LIN {X 0,Y 523.99,Z 242.839,A -85,B 0,C 180,E1 -4869.261,E2 -4869.261} C_VEL
LIN {X 0,Y 523.996,Z 242.835,A -85,B 0,C 180,E1 -4871.742,E2 -4871.742} C_VEL
LIN {X 0,Y 523.98,Z 242.844,A -85,B 0,C 180,E1 -4875.051,E2 -4875.051} C_VEL
LIN {X 0,Y 523.951,Z 242.839,A -85,B 0,C 180,E1 -4877.968,E2 -4877.968} C_VEL
LIN {X 0,Y 523.96,Z 242.841,A -85,B 0,C 180,E1 -4880.409,E2 -4880.409} C_VEL
LIN {X 0,Y 523.931,Z 242.848,A -85,B 0,C 180,E1 -4882.891,E2 -4882.891} C_VEL
LIN {X 0,Y 523.97,Z 242.839,A -85,B 0,C 180,E1 -4886.019,E2 -4886.019} C_VEL
LIN {X 0,Y 523.937,Z 242.846,A -85,B 0,C 180,E1 -4888.873,E2 -4888.873} C_VEL
LIN {X 0,Y 523.909,Z 242.843,A -85,B 0,C 180,E1 -4891.543,E2 -4891.543} C_VEL
LIN {X 0,Y 523.926,Z 242.849,A -85,B 0,C 180,E1 -4894.289,E2 -4894.289} C_VEL
LIN {X 0,Y 523.896,Z 242.849,A -85,B 0,C 180,E1 -4897.131,E2 -4897.131} C_VEL
LIN {X 0,Y 523.953,Z 242.844,A -85,B 0,C 180,E1 -4900.133,E2 -4900.133} C_VEL
LIN {X 0,Y 523.911,Z 242.846,A -85,B 0,C 180,E1 -4903.166,E2 -4903.166} C_VEL
LIN {X 0,Y 523.925,Z 242.846,A -85,B 0,C 180,E1 -4905.772,E2 -4905.772} C_VEL
LIN {X 0,Y 523.906,Z 242.848,A -85,B 0,C 180,E1 -4906.926,E2 -4906.926} C_VEL
LIN {X 0,Y 523.244,Z 242.931,A -85,B 0,C 180,E1 -4907.568,E2 -4907.568} C_VEL
LIN {X 0,Y 520.414,Z 243.286,A -85,B 0,C 180,E1 -4908.61,E2 -4908.61} C_VEL
LIN {X 0,Y 518.015,Z 243.588,A -85,B 0,C 180,E1 -4909.449,E2 -4909.449} C_VEL
LIN {X 0,Y 516.976,Z 243.717,A -85,B 0,C 180,E1 -4910.097,E2 -4910.097} C_VEL
LIN {X 0,Y 516.886,Z 243.727,A -85,B 0,C 180,E1 -4910.316,E2 -4910.316} C_VEL
LIN {X 0,Y 516.95,Z 243.891,A -85,B 0,C 180,E1 -4913.2,E2 -4913.2} C_VEL
LIN {X 0,Y 518.339,Z 251.292,A -85,B 0,C 180,E1 -4914.568,E2 -4914.568} C_VEL
LIN {X 0,Y 518.054,Z 264.877,A -85,B 0,C 180,E1 -4916.905,E2 -4916.905} C_VEL
LIN {X 0,Y 517.924,Z 268.001,A -85,B 0,C 180,E1 -4917.434,E2 -4917.434} C_VEL
LIN {X 0,Y 520.396,Z 279.84,A -85,B 0,C 180,E1 -4917.697,E2 -4917.697} C_VEL
LIN {X 0,Y 519.679,Z 404.722,A -85,B 0,C 180,E1 -4919.471,E2 -4919.471} C_VEL
LIN {X 0,Y 519.41,Z 419.428,A -85,B 0,C 180,E1 -4919.847,E2 -4919.847} C_VEL
LIN {X 0,Y 519.138,Z 432.509,A -85,B 0,C 180,E1 -4920.333,E2 -4920.333} C_VEL
LIN {X 0,Y 518.762,Z 444.641,A -85,B 0,C 180,E1 -4920.921,E2 -4920.921} C_VEL
LIN {X 0,Y 518.386,Z 456.881,A -85,B 0,C 180,E1 -4921.673,E2 -4921.673} C_VEL
LIN {X 0,Y 518.005,Z 468.213,A -85,B 0,C 180,E1 -4922.53,E2 -4922.53} C_VEL
LIN {X 0,Y 517.588,Z 479.491,A -85,B 0,C 180,E1 -4923.568,E2 -4923.568} C_VEL
LIN {X 0,Y 517.236,Z 489.292,A -85,B 0,C 180,E1 -4924.659,E2 -4924.659} C_VEL
LIN {X 0,Y 516.935,Z 498.728,A -85,B 0,C 180,E1 -4925.93,E2 -4925.93} C_VEL
LIN {X 0,Y 516.671,Z 506.432,A -85,B 0,C 180,E1 -4927.191,E2 -4927.191} C_VEL
LIN {X 0,Y 516.493,Z 512.724,A -85,B 0,C 180,E1 -4928.446,E2 -4928.446} C_VEL
LIN {X 0,Y 516.401,Z 518.527,A -85,B 0,C 180,E1 -4929.889,E2 -4929.889} C_VEL
LIN {X 0,Y 516.308,Z 522.989,A -85,B 0,C 180,E1 -4931.345,E2 -4931.345} C_VEL
LIN {X 0,Y 516.228,Z 525.75,A -85,B 0,C 180,E1 -4932.572,E2 -4932.572} C_VEL
LIN {X 0,Y 516.155,Z 528.093,A -85,B 0,C 180,E1 -4934.198,E2 -4934.198} C_VEL
LIN {X 0,Y 516.233,Z 528.801,A -85,B 0,C 180,E1 -4935.141,E2 -4935.141} C_VEL
LIN {X 0,Y 516.167,Z 528.929,A -85,B 0,C 180,E1 -4936.617,E2 -4936.617} C_VEL
LIN {X 0,Y 516.222,Z 527.753,A -85,B 0,C 180,E1 -4938.217,E2 -4938.217} C_VEL
LIN {X 0,Y 516.246,Z 525.195,A -85,B 0,C 180,E1 -4939.807,E2 -4939.807} C_VEL
LIN {X 0,Y 516.343,Z 521.175,A -85,B 0,C 180,E1 -4941.389,E2 -4941.389} C_VEL
LIN {X 0,Y 516.464,Z 515.615,A -85,B 0,C 180,E1 -4942.966,E2 -4942.966} C_VEL
LIN {X 0,Y 516.564,Z 510.366,A -85,B 0,C 180,E1 -4944.144,E2 -4944.144} C_VEL
LIN {X 0,Y 516.803,Z 502.83,A -85,B 0,C 180,E1 -4945.515,E2 -4945.515} C_VEL
LIN {X 0,Y 517.05,Z 493.564,A -85,B 0,C 180,E1 -4946.883,E2 -4946.883} C_VEL
LIN {X 0,Y 517.424,Z 483.883,A -85,B 0,C 180,E1 -4948.054,E2 -4948.054} C_VEL
LIN {X 0,Y 517.772,Z 473.197,A -85,B 0,C 180,E1 -4949.125,E2 -4949.125} C_VEL
LIN {X 0,Y 518.286,Z 461.343,A -85,B 0,C 180,E1 -4950.097,E2 -4950.097} C_VEL
LIN {X 0,Y 518.658,Z 449.737,A -85,B 0,C 180,E1 -4950.874,E2 -4950.874} C_VEL
LIN {X 0,Y 519.008,Z 437.105,A -85,B 0,C 180,E1 -4951.552,E2 -4951.552} C_VEL
LIN {X 0,Y 519.332,Z 424.209,A -85,B 0,C 180,E1 -4952.084,E2 -4952.084} C_VEL
LIN {X 0,Y 519.589,Z 410.377,A -85,B 0,C 180,E1 -4952.495,E2 -4952.495} C_VEL
LIN {X 0,Y 519.741,Z 396.025,A -85,B 0,C 180,E1 -4952.761,E2 -4952.761} C_VEL
LIN {X 0,Y 520.372,Z 279.837,A -85,B 0,C 180,E1 -4954.393,E2 -4954.393} C_VEL
LIN {X 0,Y 517.927,Z 267.832,A -85,B 0,C 180,E1 -4954.67,E2 -4954.67} C_VEL
LIN {X 0,Y 518.444,Z 251.844,A -85,B 0,C 180,E1 -4957.399,E2 -4957.399} C_VEL
LIN {X 0,Y 516.951,Z 243.718,A -85,B 0,C 180,E1 -4958.896,E2 -4958.896} C_VEL
LIN {X 0,Y 516.969,Z 243.718,A -85,B 0,C 180,E1 -4961.824,E2 -4961.824} C_VEL
LIN {X 0,Y 516.93,Z 243.719,A -85,B 0,C 180,E1 -4965.147,E2 -4965.147} C_VEL
LIN {X 0,Y 516.912,Z 243.719,A -85,B 0,C 180,E1 -4968.222,E2 -4968.222} C_VEL
LIN {X 0,Y 516.899,Z 243.718,A -85,B 0,C 180,E1 -4970.702,E2 -4970.702} C_VEL
LIN {X 0,Y 516.905,Z 243.721,A -85,B 0,C 180,E1 -4974.072,E2 -4974.072} C_VEL
LIN {X 0,Y 516.917,Z 243.715,A -85,B 0,C 180,E1 -4976.658,E2 -4976.658} C_VEL
LIN {X 0,Y 516.911,Z 243.724,A -85,B 0,C 180,E1 -4979.527,E2 -4979.527} C_VEL
LIN {X 0,Y 516.887,Z 243.719,A -85,B 0,C 180,E1 -4982.545,E2 -4982.545} C_VEL
LIN {X 0,Y 516.87,Z 243.728,A -85,B 0,C 180,E1 -4985.333,E2 -4985.333} C_VEL
LIN {X 0,Y 516.868,Z 243.724,A -85,B 0,C 180,E1 -4987.944,E2 -4987.944} C_VEL
LIN {X 0,Y 516.903,Z 243.718,A -85,B 0,C 180,E1 -4990.739,E2 -4990.739} C_VEL
LIN {X 0,Y 516.869,Z 243.723,A -85,B 0,C 180,E1 -4993.903,E2 -4993.903} C_VEL
LIN {X 0,Y 516.869,Z 243.722,A -85,B 0,C 180,E1 -4996.107,E2 -4996.107} C_VEL
LIN {X 0,Y 516.894,Z 243.727,A -85,B 0,C 180,E1 -4999.261,E2 -4999.261} C_VEL
LIN {X 0,Y 516.869,Z 243.722,A -85,B 0,C 180,E1 -5002.057,E2 -5002.057} C_VEL
LIN {X 0,Y 516.884,Z 243.728,A -85,B 0,C 180,E1 -5005.177,E2 -5005.177} C_VEL
LIN {X 0,Y 516.87,Z 243.721,A -85,B 0,C 180,E1 -5007.977,E2 -5007.977} C_VEL
LIN {X 0,Y 516.923,Z 243.719,A -85,B 0,C 180,E1 -5010.697,E2 -5010.697} C_VEL
LIN {X 0,Y 516.932,Z 243.714,A -85,B 0,C 180,E1 -5013.804,E2 -5013.804} C_VEL
LIN {X 0,Y 516.86,Z 243.73,A -85,B 0,C 180,E1 -5016.777,E2 -5016.777} C_VEL
LIN {X 0,Y 516.928,Z 243.714,A -85,B 0,C 180,E1 -5019.732,E2 -5019.732} C_VEL
LIN {X 0,Y 516.92,Z 243.721,A -85,B 0,C 180,E1 -5022.597,E2 -5022.597} C_VEL
LIN {X 0,Y 516.931,Z 243.719,A -85,B 0,C 180,E1 -5025.031,E2 -5025.031} C_VEL
LIN {X 0,Y 516.955,Z 243.713,A -85,B 0,C 180,E1 -5028.235,E2 -5028.235} C_VEL
LIN {X 0,Y 516.961,Z 243.711,A -85,B 0,C 180,E1 -5031.401,E2 -5031.401} C_VEL
LIN {X 0,Y 517.001,Z 243.705,A -85,B 0,C 180,E1 -5033.758,E2 -5033.758} C_VEL
LIN {X 0,Y 517.008,Z 243.708,A -85,B 0,C 180,E1 -5036.884,E2 -5036.884} C_VEL
LIN {X 0,Y 517.076,Z 243.698,A -85,B 0,C 180,E1 -5040.001,E2 -5040.001} C_VEL
LIN {X 0,Y 517.008,Z 243.705,A -85,B 0,C 180,E1 -5043.118,E2 -5043.118} C_VEL
LIN {X 0,Y 517.003,Z 243.712,A -85,B 0,C 180,E1 -5046.244,E2 -5046.244} C_VEL
LIN {X 0,Y 516.948,Z 243.712,A -85,B 0,C 180,E1 -5049.39,E2 -5049.39} C_VEL
LIN {X 0,Y 516.945,Z 243.715,A -85,B 0,C 180,E1 -5051.808,E2 -5051.808} C_VEL
LIN {X 0,Y 516.938,Z 243.713,A -85,B 0,C 180,E1 -5055.147,E2 -5055.147} C_VEL
LIN {X 0,Y 516.92,Z 243.723,A -85,B 0,C 180,E1 -5058.223,E2 -5058.223} C_VEL
LIN {X 0,Y 516.907,Z 243.718,A -85,B 0,C 180,E1 -5060.703,E2 -5060.703} C_VEL
LIN {X 0,Y 516.906,Z 243.726,A -85,B 0,C 180,E1 -5064.073,E2 -5064.073} C_VEL
LIN {X 0,Y 516.922,Z 243.716,A -85,B 0,C 180,E1 -5066.659,E2 -5066.659} C_VEL
LIN {X 0,Y 516.916,Z 243.719,A -85,B 0,C 180,E1 -5069.527,E2 -5069.527} C_VEL
LIN {X 0,Y 516.897,Z 243.719,A -85,B 0,C 180,E1 -5072.545,E2 -5072.545} C_VEL
LIN {X 0,Y 516.88,Z 243.722,A -85,B 0,C 180,E1 -5075.333,E2 -5075.333} C_VEL
LIN {X 0,Y 516.879,Z 243.727,A -85,B 0,C 180,E1 -5077.944,E2 -5077.944} C_VEL
LIN {X 0,Y 516.882,Z 243.72,A -85,B 0,C 180,E1 -5080.743,E2 -5080.743} C_VEL
LIN {X 0,Y 516.881,Z 243.72,A -85,B 0,C 180,E1 -5082.832,E2 -5082.832} C_VEL
LIN {X 0,Y 516.922,Z 243.716,A -85,B 0,C 180,E1 -5085.011,E2 -5085.011} C_VEL
LIN {X 0,Y 516.914,Z 243.716,A -85,B 0,C 180,E1 -5088.399,E2 -5088.399} C_VEL
LIN {X 0,Y 516.879,Z 243.725,A -85,B 0,C 180,E1 -5091.285,E2 -5091.285} C_VEL
LIN {X 0,Y 516.871,Z 243.722,A -85,B 0,C 180,E1 -5094.22,E2 -5094.22} C_VEL
LIN {X 0,Y 516.896,Z 243.721,A -85,B 0,C 180,E1 -5097.054,E2 -5097.054} C_VEL
LIN {X 0,Y 516.893,Z 243.726,A -85,B 0,C 180,E1 -5099.797,E2 -5099.797} C_VEL
LIN {X 0,Y 516.927,Z 243.719,A -85,B 0,C 180,E1 -5102.468,E2 -5102.468} C_VEL
LIN {X 0,Y 516.964,Z 243.89,A -85,B 0,C 180,E1 -5103.85,E2 -5103.85} C_VEL
LIN {X 0,Y 519.153,Z 254.919,A -85,B 0,C 180,E1 -5105.614,E2 -5105.614} C_VEL
LIN {X 0,Y 518.575,Z 273.415,A -85,B 0,C 180,E1 -5108.328,E2 -5108.328} C_VEL
LIN {X 0,Y 517.999,Z 294.61,A -85,B 0,C 180,E1 -5111.378,E2 -5111.378} C_VEL
LIN {X 0,Y 520.416,Z 308.774,A -85,B 0,C 180,E1 -5111.669,E2 -5111.669} C_VEL
LIN {X 0,Y 519.645,Z 432.714,A -85,B 0,C 180,E1 -5113.424,E2 -5113.424} C_VEL
LIN {X 0,Y 519.343,Z 447.15,A -85,B 0,C 180,E1 -5113.788,E2 -5113.788} C_VEL
LIN {X 0,Y 519.065,Z 460.688,A -85,B 0,C 180,E1 -5114.289,E2 -5114.289} C_VEL
LIN {X 0,Y 518.676,Z 472.91,A -85,B 0,C 180,E1 -5114.881,E2 -5114.881} C_VEL
LIN {X 0,Y 518.248,Z 485.767,A -85,B 0,C 180,E1 -5115.671,E2 -5115.671} C_VEL
LIN {X 0,Y 517.847,Z 497.459,A -85,B 0,C 180,E1 -5116.561,E2 -5116.561} C_VEL
LIN {X 0,Y 517.494,Z 507.19,A -85,B 0,C 180,E1 -5117.45,E2 -5117.45} C_VEL
LIN {X 0,Y 517.141,Z 517.972,A -85,B 0,C 180,E1 -5118.635,E2 -5118.635} C_VEL
LIN {X 0,Y 516.832,Z 526.875,A -85,B 0,C 180,E1 -5119.818,E2 -5119.818} C_VEL
LIN {X 0,Y 516.615,Z 535.409,A -85,B 0,C 180,E1 -5121.197,E2 -5121.197} C_VEL
LIN {X 0,Y 516.447,Z 542.287,A -85,B 0,C 180,E1 -5122.572,E2 -5122.572} C_VEL
LIN {X 0,Y 516.372,Z 547.028,A -85,B 0,C 180,E1 -5123.749,E2 -5123.749} C_VEL
LIN {X 0,Y 516.306,Z 550.868,A -85,B 0,C 180,E1 -5124.924,E2 -5124.924} C_VEL
LIN {X 0,Y 516.325,Z 553.828,A -85,B 0,C 180,E1 -5126.098,E2 -5126.098} C_VEL
LIN {X 0,Y 516.26,Z 556.535,A -85,B 0,C 180,E1 -5127.659,E2 -5127.659} C_VEL
LIN {X 0,Y 516.158,Z 557.874,A -85,B 0,C 180,E1 -5129.22,E2 -5129.22} C_VEL
LIN {X 0,Y 516.158,Z 557.873,A -85,B 0,C 180,E1 -5130.78,E2 -5130.78} C_VEL
LIN {X 0,Y 516.26,Z 556.534,A -85,B 0,C 180,E1 -5132.34,E2 -5132.34} C_VEL
LIN {X 0,Y 516.325,Z 553.826,A -85,B 0,C 180,E1 -5133.902,E2 -5133.902} C_VEL
LIN {X 0,Y 516.361,Z 549.672,A -85,B 0,C 180,E1 -5135.467,E2 -5135.467} C_VEL
LIN {X 0,Y 516.403,Z 543.949,A -85,B 0,C 180,E1 -5137.035,E2 -5137.035} C_VEL
LIN {X 0,Y 516.578,Z 537.501,A -85,B 0,C 180,E1 -5138.41,E2 -5138.41} C_VEL
LIN {X 0,Y 516.765,Z 529.489,A -85,B 0,C 180,E1 -5139.788,E2 -5139.788} C_VEL
LIN {X 0,Y 517.067,Z 521.112,A -85,B 0,C 180,E1 -5140.969,E2 -5140.969} C_VEL
LIN {X 0,Y 517.378,Z 510.785,A -85,B 0,C 180,E1 -5142.181,E2 -5142.181} C_VEL
LIN {X 0,Y 517.749,Z 499.776,A -85,B 0,C 180,E1 -5143.242,E2 -5143.242} C_VEL
LIN {X 0,Y 518.138,Z 488.589,A -85,B 0,C 180,E1 -5144.131,E2 -5144.131} C_VEL
LIN {X 0,Y 518.532,Z 476.405,A -85,B 0,C 180,E1 -5144.922,E2 -5144.922} C_VEL
LIN {X 0,Y 518.986,Z 462.889,A -85,B 0,C 180,E1 -5145.613,E2 -5145.613} C_VEL
LIN {X 0,Y 519.284,Z 448.75,A -85,B 0,C 180,E1 -5146.158,E2 -5146.158} C_VEL
LIN {X 0,Y 519.589,Z 434.929,A -85,B 0,C 180,E1 -5146.527,E2 -5146.527} C_VEL
LIN {X 0,Y 519.753,Z 412.74,A -85,B 0,C 180,E1 -5146.875,E2 -5146.875} C_VEL
LIN {X 0,Y 520.29,Z 307.794,A -85,B 0,C 180,E1 -5148.349,E2 -5148.349} C_VEL
LIN {X 0,Y 518.005,Z 294.369,A -85,B 0,C 180,E1 -5148.633,E2 -5148.633} C_VEL
LIN {X 0,Y 518.604,Z 271.897,A -85,B 0,C 180,E1 -5151.88,E2 -5151.88} C_VEL
LIN {X 0,Y 519.14,Z 254.866,A -85,B 0,C 180,E1 -5154.387,E2 -5154.387} C_VEL
LIN {X 0,Y 516.931,Z 243.722,A -85,B 0,C 180,E1 -5156.192,E2 -5156.192} C_VEL
LIN {X 0,Y 516.922,Z 243.719,A -85,B 0,C 180,E1 -5159.304,E2 -5159.304} C_VEL
LIN {X 0,Y 516.897,Z 243.726,A -85,B 0,C 180,E1 -5162.543,E2 -5162.543} C_VEL
LIN {X 0,Y 516.865,Z 243.726,A -85,B 0,C 180,E1 -5165.329,E2 -5165.329} C_VEL
LIN {X 0,Y 516.879,Z 243.724,A -85,B 0,C 180,E1 -5167.942,E2 -5167.942} C_VEL
LIN {X 0,Y 516.882,Z 243.723,A -85,B 0,C 180,E1 -5170.741,E2 -5170.741} C_VEL
LIN {X 0,Y 516.902,Z 243.721,A -85,B 0,C 180,E1 -5172.828,E2 -5172.828} C_VEL
LIN {X 0,Y 516.92,Z 243.716,A -85,B 0,C 180,E1 -5175.009,E2 -5175.009} C_VEL
LIN {X 0,Y 516.914,Z 243.723,A -85,B 0,C 180,E1 -5178.397,E2 -5178.397} C_VEL
LIN {X 0,Y 516.879,Z 243.721,A -85,B 0,C 180,E1 -5181.283,E2 -5181.283} C_VEL
LIN {X 0,Y 516.887,Z 243.718,A -85,B 0,C 180,E1 -5184.22,E2 -5184.22} C_VEL
LIN {X 0,Y 516.893,Z 243.719,A -85,B 0,C 180,E1 -5187.052,E2 -5187.052} C_VEL
LIN {X 0,Y 516.896,Z 243.723,A -85,B 0,C 180,E1 -5189.796,E2 -5189.796} C_VEL
LIN {X 0,Y 516.923,Z 243.716,A -85,B 0,C 180,E1 -5192.466,E2 -5192.466} C_VEL
LIN {X 0,Y 516.904,Z 243.718,A -85,B 0,C 180,E1 -5195.071,E2 -5195.071} C_VEL
LIN {X 0,Y 516.863,Z 243.729,A -85,B 0,C 180,E1 -5197.62,E2 -5197.62} C_VEL
LIN {X 0,Y 516.925,Z 243.717,A -85,B 0,C 180,E1 -5200.129,E2 -5200.129} C_VEL
LIN {X 0,Y 516.924,Z 243.715,A -85,B 0,C 180,E1 -5202.595,E2 -5202.595} C_VEL
LIN {X 0,Y 516.934,Z 243.714,A -85,B 0,C 180,E1 -5205.029,E2 -5205.029} C_VEL
LIN {X 0,Y 516.957,Z 243.709,A -85,B 0,C 180,E1 -5208.233,E2 -5208.233} C_VEL
LIN {X 0,Y 516.964,Z 243.718,A -85,B 0,C 180,E1 -5211.399,E2 -5211.399} C_VEL
LIN {X 0,Y 517.001,Z 243.71,A -85,B 0,C 180,E1 -5213.756,E2 -5213.756} C_VEL
LIN {X 0,Y 517.007,Z 243.706,A -85,B 0,C 180,E1 -5216.882,E2 -5216.882} C_VEL
LIN {X 0,Y 517.072,Z 243.697,A -85,B 0,C 180,E1 -5219.999,E2 -5219.999} C_VEL
LIN {X 0,Y 517.007,Z 243.711,A -85,B 0,C 180,E1 -5223.116,E2 -5223.116} C_VEL
LIN {X 0,Y 516.999,Z 243.704,A -85,B 0,C 180,E1 -5226.242,E2 -5226.242} C_VEL
LIN {X 0,Y 516.945,Z 243.715,A -85,B 0,C 180,E1 -5229.388,E2 -5229.388} C_VEL
LIN {X 0,Y 516.945,Z 243.713,A -85,B 0,C 180,E1 -5231.809,E2 -5231.809} C_VEL
LIN {X 0,Y 516.931,Z 243.721,A -85,B 0,C 180,E1 -5235.145,E2 -5235.145} C_VEL
LIN {X 0,Y 516.912,Z 243.717,A -85,B 0,C 180,E1 -5238.221,E2 -5238.221} C_VEL
LIN {X 0,Y 516.902,Z 243.724,A -85,B 0,C 180,E1 -5240.7,E2 -5240.7} C_VEL
LIN {X 0,Y 516.878,Z 243.722,A -85,B 0,C 180,E1 -5243.222,E2 -5243.222} C_VEL
LIN {X 0,Y 516.928,Z 243.717,A -85,B 0,C 180,E1 -5246.195,E2 -5246.195} C_VEL
LIN {X 0,Y 516.922,Z 243.715,A -85,B 0,C 180,E1 -5249.303,E2 -5249.303} C_VEL
LIN {X 0,Y 516.882,Z 243.727,A -85,B 0,C 180,E1 -5252.543,E2 -5252.543} C_VEL
LIN {X 0,Y 516.865,Z 243.72,A -85,B 0,C 180,E1 -5255.331,E2 -5255.331} C_VEL
LIN {X 0,Y 516.867,Z 243.726,A -85,B 0,C 180,E1 -5257.943,E2 -5257.943} C_VEL
LIN {X 0,Y 516.889,Z 243.724,A -85,B 0,C 180,E1 -5260.739,E2 -5260.739} C_VEL
LIN {X 0,Y 516.867,Z 243.727,A -85,B 0,C 180,E1 -5263.903,E2 -5263.903} C_VEL
LIN {X 0,Y 516.867,Z 243.73,A -85,B 0,C 180,E1 -5266.106,E2 -5266.106} C_VEL
LIN {X 0,Y 516.889,Z 243.722,A -85,B 0,C 180,E1 -5269.26,E2 -5269.26} C_VEL
LIN {X 0,Y 516.886,Z 243.727,A -85,B 0,C 180,E1 -5270.316,E2 -5270.316} C_VEL
LIN {X 0,Y 516.194,Z 243.813,A -85,B 0,C 180,E1 -5270.75,E2 -5270.75} C_VEL
LIN {X 0,Y 513.334,Z 244.168,A -85,B 0,C 180,E1 -5271.428,E2 -5271.428} C_VEL
LIN {X 0,Y 510.486,Z 244.526,A -85,B 0,C 180,E1 -5272.113,E2 -5272.113} C_VEL
LIN {X 0,Y 509.827,Z 244.607,A -85,B 0,C 180,E1 -5272.555,E2 -5272.555} C_VEL
LIN {X 0,Y 509.854,Z 244.69,A -85,B 0,C 180,E1 -5272.965,E2 -5272.965} C_VEL
LIN {X 0,Y 511.436,Z 252.766,A -85,B 0,C 180,E1 -5274.488,E2 -5274.488} C_VEL
LIN {X 0,Y 511.043,Z 267.316,A -85,B 0,C 180,E1 -5277.02,E2 -5277.02} C_VEL
LIN {X 0,Y 511.057,Z 268.302,A -85,B 0,C 180,E1 -5277.175,E2 -5277.175} C_VEL
LIN {X 0,Y 513.655,Z 280.569,A -85,B 0,C 180,E1 -5277.455,E2 -5277.455} C_VEL
LIN {X 0,Y 512.898,Z 405.162,A -85,B 0,C 180,E1 -5279.252,E2 -5279.252} C_VEL
LIN {X 0,Y 512.592,Z 419.721,A -85,B 0,C 180,E1 -5279.629,E2 -5279.629} C_VEL
LIN {X 0,Y 512.304,Z 432.99,A -85,B 0,C 180,E1 -5280.131,E2 -5280.131} C_VEL
LIN {X 0,Y 511.912,Z 444.924,A -85,B 0,C 180,E1 -5280.72,E2 -5280.72} C_VEL
LIN {X 0,Y 511.509,Z 456.973,A -85,B 0,C 180,E1 -5281.469,E2 -5281.469} C_VEL
LIN {X 0,Y 511.073,Z 468.458,A -85,B 0,C 180,E1 -5282.348,E2 -5282.348} C_VEL
LIN {X 0,Y 510.603,Z 480.329,A -85,B 0,C 180,E1 -5283.462,E2 -5283.462} C_VEL
LIN {X 0,Y 510.182,Z 491.265,A -85,B 0,C 180,E1 -5284.721,E2 -5284.721} C_VEL
LIN {X 0,Y 509.866,Z 500.381,A -85,B 0,C 180,E1 -5286.007,E2 -5286.007} C_VEL
LIN {X 0,Y 509.612,Z 507.829,A -85,B 0,C 180,E1 -5287.286,E2 -5287.286} C_VEL
LIN {X 0,Y 509.413,Z 513.899,A -85,B 0,C 180,E1 -5288.556,E2 -5288.556} C_VEL
LIN {X 0,Y 509.328,Z 518.789,A -85,B 0,C 180,E1 -5289.821,E2 -5289.821} C_VEL
LIN {X 0,Y 509.242,Z 522.647,A -85,B 0,C 180,E1 -5291.076,E2 -5291.076} C_VEL
LIN {X 0,Y 509.15,Z 525.583,A -85,B 0,C 180,E1 -5292.322,E2 -5292.322} C_VEL
LIN {X 0,Y 509.058,Z 528.092,A -85,B 0,C 180,E1 -5293.972,E2 -5293.972} C_VEL
LIN {X 0,Y 509.113,Z 529.158,A -85,B 0,C 180,E1 -5295.613,E2 -5295.613} C_VEL
LIN {X 0,Y 509.089,Z 528.831,A -85,B 0,C 180,E1 -5297.24,E2 -5297.24} C_VEL
LIN {X 0,Y 509.175,Z 527.124,A -85,B 0,C 180,E1 -5298.859,E2 -5298.859} C_VEL
LIN {X 0,Y 509.144,Z 524.041,A -85,B 0,C 180,E1 -5300.466,E2 -5300.466} C_VEL
LIN {X 0,Y 509.31,Z 519.482,A -85,B 0,C 180,E1 -5302.069,E2 -5302.069} C_VEL
LIN {X 0,Y 509.461,Z 513.286,A -85,B 0,C 180,E1 -5303.664,E2 -5303.664} C_VEL
LIN {X 0,Y 509.618,Z 506.418,A -85,B 0,C 180,E1 -5305.056,E2 -5305.056} C_VEL
LIN {X 0,Y 509.871,Z 497.941,A -85,B 0,C 180,E1 -5306.444,E2 -5306.444} C_VEL
LIN {X 0,Y 510.257,Z 489.099,A -85,B 0,C 180,E1 -5307.632,E2 -5307.632} C_VEL
LIN {X 0,Y 510.66,Z 478.455,A -85,B 0,C 180,E1 -5308.817,E2 -5308.817} C_VEL
LIN {X 0,Y 511.131,Z 467.685,A -85,B 0,C 180,E1 -5309.803,E2 -5309.803} C_VEL
LIN {X 0,Y 511.564,Z 455.947,A -85,B 0,C 180,E1 -5310.689,E2 -5310.689} C_VEL
LIN {X 0,Y 512.024,Z 442.98,A -85,B 0,C 180,E1 -5311.475,E2 -5311.475} C_VEL
LIN {X 0,Y 512.39,Z 429.328,A -85,B 0,C 180,E1 -5312.113,E2 -5312.113} C_VEL
LIN {X 0,Y 512.707,Z 414.894,A -85,B 0,C 180,E1 -5312.603,E2 -5312.603} C_VEL
LIN {X 0,Y 512.913,Z 400.49,A -85,B 0,C 180,E1 -5312.921,E2 -5312.921} C_VEL
LIN {X 0,Y 513.709,Z 281.236,A -85,B 0,C 180,E1 -5314.622,E2 -5314.622} C_VEL
LIN {X 0,Y 510.972,Z 268.014,A -85,B 0,C 180,E1 -5314.931,E2 -5314.931} C_VEL
LIN {X 0,Y 511.507,Z 253.142,A -85,B 0,C 180,E1 -5317.5,E2 -5317.5} C_VEL
LIN {X 0,Y 509.938,Z 244.592,A -85,B 0,C 180,E1 -5319.119,E2 -5319.119} C_VEL
LIN {X 0,Y 509.937,Z 244.595,A -85,B 0,C 180,E1 -5321.931,E2 -5321.931} C_VEL
LIN {X 0,Y 509.879,Z 244.598,A -85,B 0,C 180,E1 -5325.242,E2 -5325.242} C_VEL
LIN {X 0,Y 509.874,Z 244.599,A -85,B 0,C 180,E1 -5328.001,E2 -5328.001} C_VEL
LIN {X 0,Y 509.837,Z 244.598,A -85,B 0,C 180,E1 -5331.002,E2 -5331.002} C_VEL
LIN {X 0,Y 509.828,Z 244.605,A -85,B 0,C 180,E1 -5333.563,E2 -5333.563} C_VEL
LIN {X 0,Y 509.902,Z 244.59,A -85,B 0,C 180,E1 -5336.38,E2 -5336.38} C_VEL
LIN {X 0,Y 509.872,Z 244.594,A -85,B 0,C 180,E1 -5338.844,E2 -5338.844} C_VEL
LIN {X 0,Y 509.813,Z 244.609,A -85,B 0,C 180,E1 -5341.59,E2 -5341.59} C_VEL
LIN {X 0,Y 509.841,Z 244.597,A -85,B 0,C 180,E1 -5344.414,E2 -5344.414} C_VEL
LIN {X 0,Y 509.805,Z 244.609,A -85,B 0,C 180,E1 -5347.341,E2 -5347.341} C_VEL
LIN {X 0,Y 509.865,Z 244.594,A -85,B 0,C 180,E1 -5350.379,E2 -5350.379} C_VEL
LIN {X 0,Y 509.827,Z 244.603,A -85,B 0,C 180,E1 -5353.065,E2 -5353.065} C_VEL
LIN {X 0,Y 509.817,Z 244.602,A -85,B 0,C 180,E1 -5355.793,E2 -5355.793} C_VEL
LIN {X 0,Y 509.857,Z 244.596,A -85,B 0,C 180,E1 -5358.577,E2 -5358.577} C_VEL
LIN {X 0,Y 509.843,Z 244.598,A -85,B 0,C 180,E1 -5361.786,E2 -5361.786} C_VEL
LIN {X 0,Y 509.834,Z 244.6,A -85,B 0,C 180,E1 -5364.624,E2 -5364.624} C_VEL
LIN {X 0,Y 509.853,Z 244.599,A -85,B 0,C 180,E1 -5367.482,E2 -5367.482} C_VEL
LIN {X 0,Y 509.869,Z 244.594,A -85,B 0,C 180,E1 -5370.27,E2 -5370.27} C_VEL
LIN {X 0,Y 509.876,Z 244.601,A -85,B 0,C 180,E1 -5372.945,E2 -5372.945} C_VEL
LIN {X 0,Y 509.858,Z 244.596,A -85,B 0,C 180,E1 -5375.575,E2 -5375.575} C_VEL
LIN {X 0,Y 509.811,Z 244.601,A -85,B 0,C 180,E1 -5378.15,E2 -5378.15} C_VEL
LIN {X 0,Y 509.854,Z 244.602,A -85,B 0,C 180,E1 -5380.683,E2 -5380.683} C_VEL
LIN {X 0,Y 509.876,Z 244.596,A -85,B 0,C 180,E1 -5383.176,E2 -5383.176} C_VEL
LIN {X 0,Y 509.854,Z 244.595,A -85,B 0,C 180,E1 -5385.635,E2 -5385.635} C_VEL
LIN {X 0,Y 509.891,Z 244.592,A -85,B 0,C 180,E1 -5388.124,E2 -5388.124} C_VEL
LIN {X 0,Y 509.907,Z 244.59,A -85,B 0,C 180,E1 -5391.281,E2 -5391.281} C_VEL
LIN {X 0,Y 509.969,Z 244.581,A -85,B 0,C 180,E1 -5393.671,E2 -5393.671} C_VEL
LIN {X 0,Y 510.047,Z 244.571,A -85,B 0,C 180,E1 -5397.632,E2 -5397.632} C_VEL
LIN {X 0,Y 510.057,Z 244.574,A -85,B 0,C 180,E1 -5400.791,E2 -5400.791} C_VEL
LIN {X 0,Y 509.95,Z 244.584,A -85,B 0,C 180,E1 -5403.161,E2 -5403.161} C_VEL
LIN {X 0,Y 509.971,Z 244.589,A -85,B 0,C 180,E1 -5406.331,E2 -5406.331} C_VEL
LIN {X 0,Y 509.909,Z 244.592,A -85,B 0,C 180,E1 -5408.721,E2 -5408.721} C_VEL
LIN {X 0,Y 509.897,Z 244.594,A -85,B 0,C 180,E1 -5411.933,E2 -5411.933} C_VEL
LIN {X 0,Y 509.887,Z 244.591,A -85,B 0,C 180,E1 -5415.243,E2 -5415.243} C_VEL
LIN {X 0,Y 509.883,Z 244.598,A -85,B 0,C 180,E1 -5418.002,E2 -5418.002} C_VEL
LIN {X 0,Y 509.845,Z 244.597,A -85,B 0,C 180,E1 -5421.003,E2 -5421.003} C_VEL
LIN {X 0,Y 509.865,Z 244.597,A -85,B 0,C 180,E1 -5424.427,E2 -5424.427} C_VEL
LIN {X 0,Y 509.881,Z 244.592,A -85,B 0,C 180,E1 -5427.057,E2 -5427.057} C_VEL
LIN {X 0,Y 509.877,Z 244.598,A -85,B 0,C 180,E1 -5429.751,E2 -5429.751} C_VEL
LIN {X 0,Y 509.873,Z 244.593,A -85,B 0,C 180,E1 -5432.776,E2 -5432.776} C_VEL
LIN {X 0,Y 509.839,Z 244.602,A -85,B 0,C 180,E1 -5435.582,E2 -5435.582} C_VEL
LIN {X 0,Y 509.848,Z 244.598,A -85,B 0,C 180,E1 -5438.339,E2 -5438.339} C_VEL
LIN {X 0,Y 509.854,Z 244.6,A -85,B 0,C 180,E1 -5441.426,E2 -5441.426} C_VEL
LIN {X 0,Y 509.855,Z 244.595,A -85,B 0,C 180,E1 -5444.669,E2 -5444.669} C_VEL
LIN {X 0,Y 509.856,Z 244.597,A -85,B 0,C 180,E1 -5448.104,E2 -5448.104} C_VEL
LIN {X 0,Y 509.845,Z 244.596,A -85,B 0,C 180,E1 -5450.648,E2 -5450.648} C_VEL
LIN {X 0,Y 509.824,Z 244.606,A -85,B 0,C 180,E1 -5453.648,E2 -5453.648} C_VEL
LIN {X 0,Y 509.86,Z 244.595,A -85,B 0,C 180,E1 -5456.54,E2 -5456.54} C_VEL
LIN {X 0,Y 509.846,Z 244.606,A -85,B 0,C 180,E1 -5459.335,E2 -5459.335} C_VEL
LIN {X 0,Y 509.893,Z 244.596,A -85,B 0,C 180,E1 -5462.055,E2 -5462.055} C_VEL
LIN {X 0,Y 509.913,Z 244.693,A -85,B 0,C 180,E1 -5463.622,E2 -5463.622} C_VEL
LIN {X 0,Y 512.268,Z 256.398,A -85,B 0,C 180,E1 -5465.521,E2 -5465.521} C_VEL
LIN {X 0,Y 511.568,Z 276.065,A -85,B 0,C 180,E1 -5468.439,E2 -5468.439} C_VEL
LIN {X 0,Y 511.047,Z 294.357,A -85,B 0,C 180,E1 -5471.114,E2 -5471.114} C_VEL
LIN {X 0,Y 513.681,Z 309.516,A -85,B 0,C 180,E1 -5471.433,E2 -5471.433} C_VEL
LIN {X 0,Y 512.849,Z 432.47,A -85,B 0,C 180,E1 -5473.198,E2 -5473.198} C_VEL
LIN {X 0,Y 512.534,Z 446.636,A -85,B 0,C 180,E1 -5473.557,E2 -5473.557} C_VEL
LIN {X 0,Y 512.224,Z 460.467,A -85,B 0,C 180,E1 -5474.073,E2 -5474.073} C_VEL
LIN {X 0,Y 511.735,Z 474.464,A -85,B 0,C 180,E1 -5474.773,E2 -5474.773} C_VEL
LIN {X 0,Y 511.28,Z 486.985,A -85,B 0,C 180,E1 -5475.573,E2 -5475.573} C_VEL
LIN {X 0,Y 510.85,Z 498.427,A -85,B 0,C 180,E1 -5476.475,E2 -5476.475} C_VEL
LIN {X 0,Y 510.441,Z 509.138,A -85,B 0,C 180,E1 -5477.496,E2 -5477.496} C_VEL
LIN {X 0,Y 510.103,Z 519.403,A -85,B 0,C 180,E1 -5478.678,E2 -5478.678} C_VEL
LIN {X 0,Y 509.741,Z 528.033,A -85,B 0,C 180,E1 -5479.876,E2 -5479.876} C_VEL
LIN {X 0,Y 509.528,Z 536.301,A -85,B 0,C 180,E1 -5481.273,E2 -5481.273} C_VEL
LIN {X 0,Y 509.37,Z 542.085,A -85,B 0,C 180,E1 -5482.468,E2 -5482.468} C_VEL
LIN {X 0,Y 509.289,Z 546.828,A -85,B 0,C 180,E1 -5483.662,E2 -5483.662} C_VEL
LIN {X 0,Y 509.235,Z 550.669,A -85,B 0,C 180,E1 -5484.853,E2 -5484.853} C_VEL
LIN {X 0,Y 509.218,Z 553.628,A -85,B 0,C 180,E1 -5486.043,E2 -5486.043} C_VEL
LIN {X 0,Y 509.189,Z 556.336,A -85,B 0,C 180,E1 -5487.627,E2 -5487.627} C_VEL
LIN {X 0,Y 509.071,Z 557.675,A -85,B 0,C 180,E1 -5489.209,E2 -5489.209} C_VEL
LIN {X 0,Y 509.071,Z 557.673,A -85,B 0,C 180,E1 -5490.791,E2 -5490.791} C_VEL
LIN {X 0,Y 509.189,Z 556.334,A -85,B 0,C 180,E1 -5492.373,E2 -5492.373} C_VEL
LIN {X 0,Y 509.217,Z 553.623,A -85,B 0,C 180,E1 -5493.957,E2 -5493.957} C_VEL
LIN {X 0,Y 509.277,Z 549.468,A -85,B 0,C 180,E1 -5495.543,E2 -5495.543} C_VEL
LIN {X 0,Y 509.328,Z 543.743,A -85,B 0,C 180,E1 -5497.134,E2 -5497.134} C_VEL
LIN {X 0,Y 509.499,Z 537.292,A -85,B 0,C 180,E1 -5498.527,E2 -5498.527} C_VEL
LIN {X 0,Y 509.719,Z 529.278,A -85,B 0,C 180,E1 -5499.924,E2 -5499.924} C_VEL
LIN {X 0,Y 510.036,Z 520.899,A -85,B 0,C 180,E1 -5501.122,E2 -5501.122} C_VEL
LIN {X 0,Y 510.398,Z 510.169,A -85,B 0,C 180,E1 -5502.394,E2 -5502.394} C_VEL
LIN {X 0,Y 510.779,Z 499.556,A -85,B 0,C 180,E1 -5503.426,E2 -5503.426} C_VEL
LIN {X 0,Y 511.225,Z 488.366,A -85,B 0,C 180,E1 -5504.326,E2 -5504.326} C_VEL
LIN {X 0,Y 511.633,Z 476.176,A -85,B 0,C 180,E1 -5505.128,E2 -5505.128} C_VEL
LIN {X 0,Y 512.147,Z 462.655,A -85,B 0,C 180,E1 -5505.827,E2 -5505.827} C_VEL
LIN {X 0,Y 512.473,Z 448.51,A -85,B 0,C 180,E1 -5506.379,E2 -5506.379} C_VEL
LIN {X 0,Y 512.791,Z 434.669,A -85,B 0,C 180,E1 -5506.752,E2 -5506.752} C_VEL
LIN {X 0,Y 512.955,Z 412.454,A -85,B 0,C 180,E1 -5507.106,E2 -5507.106} C_VEL
LIN {X 0,Y 513.621,Z 309.15,A -85,B 0,C 180,E1 -5508.573,E2 -5508.573} C_VEL
LIN {X 0,Y 511.038,Z 294.168,A -85,B 0,C 180,E1 -5508.897,E2 -5508.897} C_VEL
LIN {X 0,Y 511.687,Z 273.161,A -85,B 0,C 180,E1 -5511.979,E2 -5511.979} C_VEL
LIN {X 0,Y 512.262,Z 256.444,A -85,B 0,C 180,E1 -5514.479,E2 -5514.479} C_VEL
LIN {X 0,Y 510.248,Z 246.262,A -85,B 0,C 180,E1 -5516.151,E2 -5516.151} C_VEL
LIN {X 0,Y 509.886,Z 244.598,A -85,B 0,C 180,E1 -5516.435,E2 -5516.435} C_VEL
LIN {X 0,Y 509.877,Z 244.599,A -85,B 0,C 180,E1 -5518.843,E2 -5518.843} C_VEL
LIN {X 0,Y 509.821,Z 244.604,A -85,B 0,C 180,E1 -5521.589,E2 -5521.589} C_VEL
LIN {X 0,Y 509.847,Z 244.605,A -85,B 0,C 180,E1 -5524.413,E2 -5524.413} C_VEL
LIN {X 0,Y 509.815,Z 244.602,A -85,B 0,C 180,E1 -5527.34,E2 -5527.34} C_VEL
LIN {X 0,Y 509.836,Z 244.603,A -85,B 0,C 180,E1 -5530.381,E2 -5530.381} C_VEL
LIN {X 0,Y 509.837,Z 244.599,A -85,B 0,C 180,E1 -5533.063,E2 -5533.063} C_VEL
LIN {X 0,Y 509.828,Z 244.602,A -85,B 0,C 180,E1 -5535.791,E2 -5535.791} C_VEL
LIN {X 0,Y 509.855,Z 244.6,A -85,B 0,C 180,E1 -5538.574,E2 -5538.574} C_VEL
LIN {X 0,Y 509.848,Z 244.601,A -85,B 0,C 180,E1 -5541.785,E2 -5541.785} C_VEL
LIN {X 0,Y 509.842,Z 244.593,A -85,B 0,C 180,E1 -5544.622,E2 -5544.622} C_VEL
LIN {X 0,Y 509.861,Z 244.597,A -85,B 0,C 180,E1 -5547.48,E2 -5547.48} C_VEL
LIN {X 0,Y 509.876,Z 244.597,A -85,B 0,C 180,E1 -5550.268,E2 -5550.268} C_VEL
LIN {X 0,Y 509.88,Z 244.591,A -85,B 0,C 180,E1 -5552.943,E2 -5552.943} C_VEL
LIN {X 0,Y 509.863,Z 244.6,A -85,B 0,C 180,E1 -5555.573,E2 -5555.573} C_VEL
LIN {X 0,Y 509.843,Z 244.598,A -85,B 0,C 180,E1 -5558.997,E2 -5558.997} C_VEL
LIN {X 0,Y 509.881,Z 244.597,A -85,B 0,C 180,E1 -5561.998,E2 -5561.998} C_VEL
LIN {X 0,Y 509.902,Z 244.589,A -85,B 0,C 180,E1 -5564.818,E2 -5564.818} C_VEL
LIN {X 0,Y 509.897,Z 244.589,A -85,B 0,C 180,E1 -5568.12,E2 -5568.12} C_VEL
LIN {X 0,Y 509.91,Z 244.595,A -85,B 0,C 180,E1 -5571.279,E2 -5571.279} C_VEL
LIN {X 0,Y 509.969,Z 244.587,A -85,B 0,C 180,E1 -5573.669,E2 -5573.669} C_VEL
LIN {X 0,Y 510.045,Z 244.576,A -85,B 0,C 180,E1 -5577.63,E2 -5577.63} C_VEL
LIN {X 0,Y 510.044,Z 244.572,A -85,B 0,C 180,E1 -5579.999,E2 -5579.999} C_VEL
LIN {X 0,Y 510.044,Z 244.571,A -85,B 0,C 180,E1 -5582.368,E2 -5582.368} C_VEL
LIN {X 0,Y 509.967,Z 244.58,A -85,B 0,C 180,E1 -5586.329,E2 -5586.329} C_VEL
LIN {X 0,Y 509.906,Z 244.593,A -85,B 0,C 180,E1 -5588.719,E2 -5588.719} C_VEL
LIN {X 0,Y 509.893,Z 244.591,A -85,B 0,C 180,E1 -5591.931,E2 -5591.931} C_VEL
LIN {X 0,Y 509.881,Z 244.597,A -85,B 0,C 180,E1 -5595.241,E2 -5595.241} C_VEL
LIN {X 0,Y 509.875,Z 244.592,A -85,B 0,C 180,E1 -5598,E2 -5598} C_VEL
LIN {X 0,Y 509.844,Z 244.603,A -85,B 0,C 180,E1 -5601.001,E2 -5601.001} C_VEL
LIN {X 0,Y 509.837,Z 244.597,A -85,B 0,C 180,E1 -5603.562,E2 -5603.562} C_VEL
LIN {X 0,Y 509.897,Z 244.595,A -85,B 0,C 180,E1 -5606.378,E2 -5606.378} C_VEL
LIN {X 0,Y 509.871,Z 244.598,A -85,B 0,C 180,E1 -5608.843,E2 -5608.843} C_VEL
LIN {X 0,Y 509.807,Z 244.599,A -85,B 0,C 180,E1 -5611.589,E2 -5611.589} C_VEL
LIN {X 0,Y 509.837,Z 244.603,A -85,B 0,C 180,E1 -5614.413,E2 -5614.413} C_VEL
LIN {X 0,Y 509.804,Z 244.604,A -85,B 0,C 180,E1 -5617.34,E2 -5617.34} C_VEL
LIN {X 0,Y 509.846,Z 244.605,A -85,B 0,C 180,E1 -5620.379,E2 -5620.379} C_VEL
LIN {X 0,Y 509.825,Z 244.602,A -85,B 0,C 180,E1 -5623.064,E2 -5623.064} C_VEL
LIN {X 0,Y 509.815,Z 244.604,A -85,B 0,C 180,E1 -5625.792,E2 -5625.792} C_VEL
LIN {X 0,Y 509.85,Z 244.601,A -85,B 0,C 180,E1 -5628.575,E2 -5628.575} C_VEL
LIN {X 0,Y 509.837,Z 244.606,A -85,B 0,C 180,E1 -5631.786,E2 -5631.786} C_VEL
LIN {X 0,Y 509.827,Z 244.607,A -85,B 0,C 180,E1 -5632.555,E2 -5632.555} C_VEL
LIN {X 0,Y 509.606,Z 245.452,A -85,B 0,C 180,E1 -5632.993,E2 -5632.993} C_VEL
LIN {X 0,Y 508.631,Z 248.512,A -85,B 0,C 180,E1 -5633.585,E2 -5633.585} C_VEL
LIN {X 0,Y 504.714,Z 258.723,A -85,B 0,C 180,E1 -5635.203,E2 -5635.203} C_VEL
LIN {X 0,Y 504.401,Z 260.877,A -85,B 0,C 180,E1 -5635.579,E2 -5635.579} C_VEL
LIN {X 0,Y 504.113,Z 268.425,A -85,B 0,C 180,E1 -5636.9,E2 -5636.9} C_VEL
LIN {X 0,Y 507.004,Z 282.177,A -85,B 0,C 180,E1 -5637.22,E2 -5637.22} C_VEL
LIN {X 0,Y 506.135,Z 404.315,A -85,B 0,C 180,E1 -5638.999,E2 -5638.999} C_VEL
LIN {X 0,Y 505.86,Z 418.709,A -85,B 0,C 180,E1 -5639.364,E2 -5639.364} C_VEL
LIN {X 0,Y 505.556,Z 431.398,A -85,B 0,C 180,E1 -5639.831,E2 -5639.831} C_VEL
LIN {X 0,Y 505.151,Z 443.282,A -85,B 0,C 180,E1 -5640.404,E2 -5640.404} C_VEL
LIN {X 0,Y 504.649,Z 456.791,A -85,B 0,C 180,E1 -5641.24,E2 -5641.24} C_VEL
LIN {X 0,Y 504.15,Z 468.704,A -85,B 0,C 180,E1 -5642.161,E2 -5642.161} C_VEL
LIN {X 0,Y 503.656,Z 480.24,A -85,B 0,C 180,E1 -5643.256,E2 -5643.256} C_VEL
LIN {X 0,Y 503.306,Z 489.767,A -85,B 0,C 180,E1 -5644.351,E2 -5644.351} C_VEL
LIN {X 0,Y 502.915,Z 499.186,A -85,B 0,C 180,E1 -5645.655,E2 -5645.655} C_VEL
LIN {X 0,Y 502.61,Z 506.883,A -85,B 0,C 180,E1 -5646.951,E2 -5646.951} C_VEL
LIN {X 0,Y 502.397,Z 513.167,A -85,B 0,C 180,E1 -5648.241,E2 -5648.241} C_VEL
LIN {X 0,Y 502.259,Z 518.639,A -85,B 0,C 180,E1 -5649.633,E2 -5649.633} C_VEL
LIN {X 0,Y 502.151,Z 523.416,A -85,B 0,C 180,E1 -5651.222,E2 -5651.222} C_VEL
LIN {X 0,Y 502.068,Z 525.542,A -85,B 0,C 180,E1 -5652.146,E2 -5652.146} C_VEL
LIN {X 0,Y 501.988,Z 528.088,A -85,B 0,C 180,E1 -5653.74,E2 -5653.74} C_VEL
LIN {X 0,Y 502.041,Z 529.318,A -85,B 0,C 180,E1 -5655.406,E2 -5655.406} C_VEL
LIN {X 0,Y 501.986,Z 529.15,A -85,B 0,C 180,E1 -5657.056,E2 -5657.056} C_VEL
LIN {X 0,Y 502.071,Z 527.6,A -85,B 0,C 180,E1 -5658.699,E2 -5658.699} C_VEL
LIN {X 0,Y 502.052,Z 524.675,A -85,B 0,C 180,E1 -5660.33,E2 -5660.33} C_VEL
LIN {X 0,Y 502.214,Z 520.295,A -85,B 0,C 180,E1 -5661.956,E2 -5661.956} C_VEL
LIN {X 0,Y 502.384,Z 514.352,A -85,B 0,C 180,E1 -5663.575,E2 -5663.575} C_VEL
LIN {X 0,Y 502.549,Z 507.69,A -85,B 0,C 180,E1 -5664.986,E2 -5664.986} C_VEL
LIN {X 0,Y 502.843,Z 499.432,A -85,B 0,C 180,E1 -5666.394,E2 -5666.394} C_VEL
LIN {X 0,Y 503.205,Z 490.856,A -85,B 0,C 180,E1 -5667.599,E2 -5667.599} C_VEL
LIN {X 0,Y 503.649,Z 480.509,A -85,B 0,C 180,E1 -5668.801,E2 -5668.801} C_VEL
LIN {X 0,Y 504.166,Z 468.968,A -85,B 0,C 180,E1 -5669.9,E2 -5669.9} C_VEL
LIN {X 0,Y 504.63,Z 457.456,A -85,B 0,C 180,E1 -5670.798,E2 -5670.798} C_VEL
LIN {X 0,Y 505.123,Z 444.816,A -85,B 0,C 180,E1 -5671.595,E2 -5671.595} C_VEL
LIN {X 0,Y 505.553,Z 431.725,A -85,B 0,C 180,E1 -5672.241,E2 -5672.241} C_VEL
LIN {X 0,Y 505.884,Z 417.511,A -85,B 0,C 180,E1 -5672.762,E2 -5672.762} C_VEL
LIN {X 0,Y 506.095,Z 403.248,A -85,B 0,C 180,E1 -5673.11,E2 -5673.11} C_VEL
LIN {X 0,Y 506.941,Z 281.909,A -85,B 0,C 180,E1 -5674.871,E2 -5674.871} C_VEL
LIN {X 0,Y 504.072,Z 268.187,A -85,B 0,C 180,E1 -5675.2,E2 -5675.2} C_VEL
LIN {X 0,Y 504.587,Z 254.441,A -85,B 0,C 180,E1 -5677.603,E2 -5677.603} C_VEL
LIN {X 0,Y 502.867,Z 245.473,A -85,B 0,C 180,E1 -5679.299,E2 -5679.299} C_VEL
LIN {X 0,Y 502.88,Z 245.474,A -85,B 0,C 180,E1 -5682.101,E2 -5682.101} C_VEL
LIN {X 0,Y 502.834,Z 245.478,A -85,B 0,C 180,E1 -5685.4,E2 -5685.4} C_VEL
LIN {X 0,Y 502.832,Z 245.474,A -85,B 0,C 180,E1 -5688.123,E2 -5688.123} C_VEL
LIN {X 0,Y 502.814,Z 245.473,A -85,B 0,C 180,E1 -5690.537,E2 -5690.537} C_VEL
LIN {X 0,Y 502.784,Z 245.482,A -85,B 0,C 180,E1 -5693.914,E2 -5693.914} C_VEL
LIN {X 0,Y 502.867,Z 245.466,A -85,B 0,C 180,E1 -5696.565,E2 -5696.565} C_VEL
LIN {X 0,Y 502.825,Z 245.475,A -85,B 0,C 180,E1 -5699.287,E2 -5699.287} C_VEL
LIN {X 0,Y 502.775,Z 245.479,A -85,B 0,C 180,E1 -5702.085,E2 -5702.085} C_VEL
LIN {X 0,Y 502.796,Z 245.477,A -85,B 0,C 180,E1 -5704.965,E2 -5704.965} C_VEL
LIN {X 0,Y 502.783,Z 245.478,A -85,B 0,C 180,E1 -5707.954,E2 -5707.954} C_VEL
LIN {X 0,Y 502.818,Z 245.476,A -85,B 0,C 180,E1 -5711.065,E2 -5711.065} C_VEL
LIN {X 0,Y 502.77,Z 245.486,A -85,B 0,C 180,E1 -5713.377,E2 -5713.377} C_VEL
LIN {X 0,Y 502.776,Z 245.481,A -85,B 0,C 180,E1 -5715.662,E2 -5715.662} C_VEL
LIN {X 0,Y 502.825,Z 245.472,A -85,B 0,C 180,E1 -5717.866,E2 -5717.866} C_VEL
LIN {X 0,Y 502.808,Z 245.479,A -85,B 0,C 180,E1 -5721.027,E2 -5721.027} C_VEL
LIN {X 0,Y 502.773,Z 245.477,A -85,B 0,C 180,E1 -5724.168,E2 -5724.168} C_VEL
LIN {X 0,Y 502.82,Z 245.479,A -85,B 0,C 180,E1 -5726.994,E2 -5726.994} C_VEL
LIN {X 0,Y 502.818,Z 245.472,A -85,B 0,C 180,E1 -5730.062,E2 -5730.062} C_VEL
LIN {X 0,Y 502.823,Z 245.474,A -85,B 0,C 180,E1 -5732.534,E2 -5732.534} C_VEL
LIN {X 0,Y 502.817,Z 245.476,A -85,B 0,C 180,E1 -5735.299,E2 -5735.299} C_VEL
LIN {X 0,Y 502.773,Z 245.477,A -85,B 0,C 180,E1 -5737.828,E2 -5737.828} C_VEL
LIN {X 0,Y 502.815,Z 245.475,A -85,B 0,C 180,E1 -5740.401,E2 -5740.401} C_VEL
LIN {X 0,Y 502.826,Z 245.478,A -85,B 0,C 180,E1 -5742.933,E2 -5742.933} C_VEL
LIN {X 0,Y 502.834,Z 245.471,A -85,B 0,C 180,E1 -5745.43,E2 -5745.43} C_VEL
LIN {X 0,Y 502.867,Z 245.474,A -85,B 0,C 180,E1 -5748.718,E2 -5748.718} C_VEL
LIN {X 0,Y 502.892,Z 245.464,A -85,B 0,C 180,E1 -5751.968,E2 -5751.968} C_VEL
LIN {X 0,Y 502.938,Z 245.463,A -85,B 0,C 180,E1 -5754.388,E2 -5754.388} C_VEL
LIN {X 0,Y 503.017,Z 245.447,A -85,B 0,C 180,E1 -5757.599,E2 -5757.599} C_VEL
LIN {X 0,Y 503.018,Z 245.449,A -85,B 0,C 180,E1 -5760.001,E2 -5760.001} C_VEL
LIN {X 0,Y 503.017,Z 245.455,A -85,B 0,C 180,E1 -5762.403,E2 -5762.403} C_VEL
LIN {X 0,Y 502.931,Z 245.458,A -85,B 0,C 180,E1 -5765.615,E2 -5765.615} C_VEL
LIN {X 0,Y 502.895,Z 245.467,A -85,B 0,C 180,E1 -5768.034,E2 -5768.034} C_VEL
LIN {X 0,Y 502.87,Z 245.465,A -85,B 0,C 180,E1 -5771.284,E2 -5771.284} C_VEL
LIN {X 0,Y 502.839,Z 245.473,A -85,B 0,C 180,E1 -5774.572,E2 -5774.572} C_VEL
LIN {X 0,Y 502.856,Z 245.472,A -85,B 0,C 180,E1 -5777.908,E2 -5777.908} C_VEL
LIN {X 0,Y 502.823,Z 245.474,A -85,B 0,C 180,E1 -5780.537,E2 -5780.537} C_VEL
LIN {X 0,Y 502.789,Z 245.475,A -85,B 0,C 180,E1 -5783.042,E2 -5783.042} C_VEL
LIN {X 0,Y 502.836,Z 245.474,A -85,B 0,C 180,E1 -5785.677,E2 -5785.677} C_VEL
LIN {X 0,Y 502.837,Z 245.473,A -85,B 0,C 180,E1 -5788.374,E2 -5788.374} C_VEL
LIN {X 0,Y 502.794,Z 245.478,A -85,B 0,C 180,E1 -5791.501,E2 -5791.501} C_VEL
LIN {X 0,Y 502.803,Z 245.475,A -85,B 0,C 180,E1 -5794.446,E2 -5794.446} C_VEL
LIN {X 0,Y 502.779,Z 245.478,A -85,B 0,C 180,E1 -5797.179,E2 -5797.179} C_VEL
LIN {X 0,Y 502.786,Z 245.481,A -85,B 0,C 180,E1 -5800.016,E2 -5800.016} C_VEL
LIN {X 0,Y 502.801,Z 245.476,A -85,B 0,C 180,E1 -5802.2,E2 -5802.2} C_VEL
LIN {X 0,Y 502.8,Z 245.48,A -85,B 0,C 180,E1 -5805.469,E2 -5805.469} C_VEL
LIN {X 0,Y 502.819,Z 245.473,A -85,B 0,C 180,E1 -5808.935,E2 -5808.935} C_VEL
LIN {X 0,Y 502.792,Z 245.477,A -85,B 0,C 180,E1 -5812.047,E2 -5812.047} C_VEL
LIN {X 0,Y 502.799,Z 245.477,A -85,B 0,C 180,E1 -5815.035,E2 -5815.035} C_VEL
LIN {X 0,Y 502.785,Z 245.483,A -85,B 0,C 180,E1 -5817.916,E2 -5817.916} C_VEL
LIN {X 0,Y 502.825,Z 245.476,A -85,B 0,C 180,E1 -5820.713,E2 -5820.713} C_VEL
LIN {X 0,Y 502.889,Z 245.626,A -85,B 0,C 180,E1 -5823.413,E2 -5823.413} C_VEL
LIN {X 0,Y 505.317,Z 257.305,A -85,B 0,C 180,E1 -5825.34,E2 -5825.34} C_VEL
LIN {X 0,Y 504.926,Z 270.154,A -85,B 0,C 180,E1 -5827.279,E2 -5827.279} C_VEL
LIN {X 0,Y 504.158,Z 292.915,A -85,B 0,C 180,E1 -5830.666,E2 -5830.666} C_VEL
LIN {X 0,Y 504.088,Z 294.105,A -85,B 0,C 180,E1 -5830.841,E2 -5830.841} C_VEL
LIN {X 0,Y 506.946,Z 311.221,A -85,B 0,C 180,E1 -5831.206,E2 -5831.206} C_VEL
LIN {X 0,Y 506.059,Z 432.225,A -85,B 0,C 180,E1 -5832.966,E2 -5832.966} C_VEL
LIN {X 0,Y 505.713,Z 446.284,A -85,B 0,C 180,E1 -5833.325,E2 -5833.325} C_VEL
LIN {X 0,Y 505.448,Z 459.009,A -85,B 0,C 180,E1 -5833.797,E2 -5833.797} C_VEL
LIN {X 0,Y 504.914,Z 472.477,A -85,B 0,C 180,E1 -5834.458,E2 -5834.458} C_VEL
LIN {X 0,Y 504.435,Z 485.342,A -85,B 0,C 180,E1 -5835.27,E2 -5835.27} C_VEL
LIN {X 0,Y 503.916,Z 497.037,A -85,B 0,C 180,E1 -5836.182,E2 -5836.182} C_VEL
LIN {X 0,Y 503.468,Z 507.851,A -85,B 0,C 180,E1 -5837.207,E2 -5837.207} C_VEL
LIN {X 0,Y 503.118,Z 517.627,A -85,B 0,C 180,E1 -5838.322,E2 -5838.322} C_VEL
LIN {X 0,Y 502.802,Z 526.468,A -85,B 0,C 180,E1 -5839.531,E2 -5839.531} C_VEL
LIN {X 0,Y 502.491,Z 535.004,A -85,B 0,C 180,E1 -5840.947,E2 -5840.947} C_VEL
LIN {X 0,Y 502.294,Z 541.884,A -85,B 0,C 180,E1 -5842.362,E2 -5842.362} C_VEL
LIN {X 0,Y 502.216,Z 546.628,A -85,B 0,C 180,E1 -5843.572,E2 -5843.572} C_VEL
LIN {X 0,Y 502.165,Z 550.47,A -85,B 0,C 180,E1 -5844.781,E2 -5844.781} C_VEL
LIN {X 0,Y 502.112,Z 553.428,A -85,B 0,C 180,E1 -5845.987,E2 -5845.987} C_VEL
LIN {X 0,Y 502.09,Z 556.137,A -85,B 0,C 180,E1 -5847.593,E2 -5847.593} C_VEL
LIN {X 0,Y 501.988,Z 557.476,A -85,B 0,C 180,E1 -5849.198,E2 -5849.198} C_VEL
LIN {X 0,Y 501.988,Z 557.474,A -85,B 0,C 180,E1 -5850.802,E2 -5850.802} C_VEL
LIN {X 0,Y 502.09,Z 556.133,A -85,B 0,C 180,E1 -5852.407,E2 -5852.407} C_VEL
LIN {X 0,Y 502.112,Z 553.42,A -85,B 0,C 180,E1 -5854.013,E2 -5854.013} C_VEL
LIN {X 0,Y 502.193,Z 549.263,A -85,B 0,C 180,E1 -5855.622,E2 -5855.622} C_VEL
LIN {X 0,Y 502.254,Z 543.536,A -85,B 0,C 180,E1 -5857.235,E2 -5857.235} C_VEL
LIN {X 0,Y 502.422,Z 537.083,A -85,B 0,C 180,E1 -5858.648,E2 -5858.648} C_VEL
LIN {X 0,Y 502.673,Z 529.067,A -85,B 0,C 180,E1 -5860.065,E2 -5860.065} C_VEL
LIN {X 0,Y 503.014,Z 520.685,A -85,B 0,C 180,E1 -5861.28,E2 -5861.28} C_VEL
LIN {X 0,Y 503.359,Z 510.952,A -85,B 0,C 180,E1 -5862.457,E2 -5862.457} C_VEL
LIN {X 0,Y 503.771,Z 500.441,A -85,B 0,C 180,E1 -5863.513,E2 -5863.513} C_VEL
LIN {X 0,Y 504.297,Z 488.141,A -85,B 0,C 180,E1 -5864.528,E2 -5864.528} C_VEL
LIN {X 0,Y 504.75,Z 475.948,A -85,B 0,C 180,E1 -5865.34,E2 -5865.34} C_VEL
LIN {X 0,Y 505.299,Z 462.421,A -85,B 0,C 180,E1 -5866.047,E2 -5866.047} C_VEL
LIN {X 0,Y 505.674,Z 448.331,A -85,B 0,C 180,E1 -5866.603,E2 -5866.603} C_VEL
LIN {X 0,Y 505.971,Z 434.414,A -85,B 0,C 180,E1 -5866.985,E2 -5866.985} C_VEL
LIN {X 0,Y 506.195,Z 412.209,A -85,B 0,C 180,E1 -5867.341,E2 -5867.341} C_VEL
LIN {X 0,Y 506.915,Z 310.28,A -85,B 0,C 180,E1 -5868.809,E2 -5868.809} C_VEL
LIN {X 0,Y 504.113,Z 293.989,A -85,B 0,C 180,E1 -5869.165,E2 -5869.165} C_VEL
LIN {X 0,Y 504.799,Z 273.02,A -85,B 0,C 180,E1 -5872.295,E2 -5872.295} C_VEL
LIN {X 0,Y 505.356,Z 258.907,A -85,B 0,C 180,E1 -5874.439,E2 -5874.439} C_VEL
LIN {X 0,Y 504.785,Z 254.336,A -85,B 0,C 180,E1 -5875.179,E2 -5875.179} C_VEL
LIN {X 0,Y 502.852,Z 245.475,A -85,B 0,C 180,E1 -5876.717,E2 -5876.717} C_VEL
LIN {X 0,Y 502.824,Z 245.476,A -85,B 0,C 180,E1 -5879.287,E2 -5879.287} C_VEL
LIN {X 0,Y 502.785,Z 245.484,A -85,B 0,C 180,E1 -5882.084,E2 -5882.084} C_VEL
LIN {X 0,Y 502.798,Z 245.482,A -85,B 0,C 180,E1 -5884.965,E2 -5884.965} C_VEL
LIN {X 0,Y 502.791,Z 245.479,A -85,B 0,C 180,E1 -5887.953,E2 -5887.953} C_VEL
LIN {X 0,Y 502.818,Z 245.472,A -85,B 0,C 180,E1 -5891.065,E2 -5891.065} C_VEL
LIN {X 0,Y 502.779,Z 245.478,A -85,B 0,C 180,E1 -5893.375,E2 -5893.375} C_VEL
LIN {X 0,Y 502.787,Z 245.478,A -85,B 0,C 180,E1 -5895.66,E2 -5895.66} C_VEL
LIN {X 0,Y 502.816,Z 245.474,A -85,B 0,C 180,E1 -5899.004,E2 -5899.004} C_VEL
LIN {X 0,Y 502.79,Z 245.483,A -85,B 0,C 180,E1 -5902.045,E2 -5902.045} C_VEL
LIN {X 0,Y 502.805,Z 245.468,A -85,B 0,C 180,E1 -5905.034,E2 -5905.034} C_VEL
LIN {X 0,Y 502.783,Z 245.484,A -85,B 0,C 180,E1 -5907.915,E2 -5907.915} C_VEL
LIN {X 0,Y 502.832,Z 245.471,A -85,B 0,C 180,E1 -5910.712,E2 -5910.712} C_VEL
LIN {X 0,Y 502.857,Z 245.469,A -85,B 0,C 180,E1 -5913.438,E2 -5913.438} C_VEL
LIN {X 0,Y 502.785,Z 245.48,A -85,B 0,C 180,E1 -5916.085,E2 -5916.085} C_VEL
LIN {X 0,Y 502.776,Z 245.477,A -85,B 0,C 180,E1 -5918.688,E2 -5918.688} C_VEL
LIN {X 0,Y 502.823,Z 245.473,A -85,B 0,C 180,E1 -5921.247,E2 -5921.247} C_VEL
LIN {X 0,Y 502.817,Z 245.476,A -85,B 0,C 180,E1 -5923.766,E2 -5923.766} C_VEL
LIN {X 0,Y 502.824,Z 245.473,A -85,B 0,C 180,E1 -5926.254,E2 -5926.254} C_VEL
LIN {X 0,Y 502.873,Z 245.463,A -85,B 0,C 180,E1 -5928.716,E2 -5928.716} C_VEL
LIN {X 0,Y 502.894,Z 245.462,A -85,B 0,C 180,E1 -5931.966,E2 -5931.966} C_VEL
LIN {X 0,Y 502.931,Z 245.459,A -85,B 0,C 180,E1 -5934.385,E2 -5934.385} C_VEL
LIN {X 0,Y 503.015,Z 245.452,A -85,B 0,C 180,E1 -5937.597,E2 -5937.597} C_VEL
LIN {X 0,Y 503.015,Z 245.448,A -85,B 0,C 180,E1 -5939.999,E2 -5939.999} C_VEL
LIN {X 0,Y 503.014,Z 245.447,A -85,B 0,C 180,E1 -5942.401,E2 -5942.401} C_VEL
LIN {X 0,Y 502.928,Z 245.459,A -85,B 0,C 180,E1 -5945.612,E2 -5945.612} C_VEL
LIN {X 0,Y 502.89,Z 245.464,A -85,B 0,C 180,E1 -5948.032,E2 -5948.032} C_VEL
LIN {X 0,Y 502.87,Z 245.471,A -85,B 0,C 180,E1 -5951.282,E2 -5951.282} C_VEL
LIN {X 0,Y 502.832,Z 245.472,A -85,B 0,C 180,E1 -5954.57,E2 -5954.57} C_VEL
LIN {X 0,Y 502.849,Z 245.467,A -85,B 0,C 180,E1 -5957.906,E2 -5957.906} C_VEL
LIN {X 0,Y 502.817,Z 245.477,A -85,B 0,C 180,E1 -5960.536,E2 -5960.536} C_VEL
LIN {X 0,Y 502.793,Z 245.479,A -85,B 0,C 180,E1 -5963.039,E2 -5963.039} C_VEL
LIN {X 0,Y 502.827,Z 245.472,A -85,B 0,C 180,E1 -5965.675,E2 -5965.675} C_VEL
LIN {X 0,Y 502.828,Z 245.476,A -85,B 0,C 180,E1 -5968.372,E2 -5968.372} C_VEL
LIN {X 0,Y 502.779,Z 245.475,A -85,B 0,C 180,E1 -5971.498,E2 -5971.498} C_VEL
LIN {X 0,Y 502.79,Z 245.48,A -85,B 0,C 180,E1 -5974.444,E2 -5974.444} C_VEL
LIN {X 0,Y 502.766,Z 245.481,A -85,B 0,C 180,E1 -5977.178,E2 -5977.178} C_VEL
LIN {X 0,Y 502.807,Z 245.476,A -85,B 0,C 180,E1 -5980.011,E2 -5980.011} C_VEL
LIN {X 0,Y 502.808,Z 245.478,A -85,B 0,C 180,E1 -5982.201,E2 -5982.201} C_VEL
LIN {X 0,Y 502.785,Z 245.478,A -85,B 0,C 180,E1 -5985.468,E2 -5985.468} C_VEL
LIN {X 0,Y 502.814,Z 245.478,A -85,B 0,C 180,E1 -5987.864,E2 -5987.864} C_VEL
LIN {X 0,Y 502.794,Z 245.482,A -85,B 0,C 180,E1 -5991.024,E2 -5991.024} C_VEL
LIN {X 0,Y 502.801,Z 245.524,A -85,B 0,C 180,E1 -5992.727,E2 -5992.727} C_VEL
LIN {X 0,Y 504.571,Z 254.483,A -85,B 0,C 180,E1 -5994.443,E2 -5994.443} C_VEL
LIN {X 0,Y 504.401,Z 260.877,A -85,B 0,C 180,E1 -5995.579,E2 -5995.579} C_VEL
LIN {X 0,Y 503.728,Z 263.403,A -85,B 0,C 180,E1 -5995.941,E2 -5995.941} C_VEL
LIN {X 0,Y 502.32,Z 266.347,A -85,B 0,C 180,E1 -5996.238,E2 -5996.238} C_VEL
LIN {X 0,Y 500.278,Z 270.755,A -85,B 0,C 180,E1 -5996.547,E2 -5996.547} C_VEL
LIN {X 0,Y 499.183,Z 275.07,A -85,B 0,C 180,E1 -5996.749,E2 -5996.749} C_VEL
LIN {X 0,Y 499.333,Z 278.316,A -85,B 0,C 180,E1 -5996.85,E2 -5996.85} C_VEL
LIN {X 0,Y 500.319,Z 283.574,A -85,B 0,C 180,E1 -5996.97,E2 -5996.97} C_VEL
LIN {X 0,Y 499.346,Z 405.708,A -85,B 0,C 180,E1 -5998.783,E2 -5998.783} C_VEL
LIN {X 0,Y 499.044,Z 419.892,A -85,B 0,C 180,E1 -5999.16,E2 -5999.16} C_VEL
LIN {X 0,Y 498.675,Z 433.501,A -85,B 0,C 180,E1 -5999.688,E2 -5999.688} C_VEL
LIN {X 0,Y 498.22,Z 445.523,A -85,B 0,C 180,E1 -6000.299,E2 -6000.299} C_VEL
LIN {X 0,Y 497.729,Z 457.893,A -85,B 0,C 180,E1 -6001.094,E2 -6001.094} C_VEL
LIN {X 0,Y 497.181,Z 470.23,A -85,B 0,C 180,E1 -6002.08,E2 -6002.08} C_VEL
LIN {X 0,Y 496.679,Z 481.051,A -85,B 0,C 180,E1 -6003.138,E2 -6003.138} C_VEL
LIN {X 0,Y 496.234,Z 491.738,A -85,B 0,C 180,E1 -6004.409,E2 -6004.409} C_VEL
LIN {X 0,Y 495.827,Z 500.833,A -85,B 0,C 180,E1 -6005.73,E2 -6005.73} C_VEL
LIN {X 0,Y 495.496,Z 509.071,A -85,B 0,C 180,E1 -6007.207,E2 -6007.207} C_VEL
LIN {X 0,Y 495.31,Z 514.342,A -85,B 0,C 180,E1 -6008.352,E2 -6008.352} C_VEL
LIN {X 0,Y 495.183,Z 518.705,A -85,B 0,C 180,E1 -6009.503,E2 -6009.503} C_VEL
LIN {X 0,Y 495.087,Z 523.075,A -85,B 0,C 180,E1 -6010.944,E2 -6010.944} C_VEL
LIN {X 0,Y 494.999,Z 525.619,A -85,B 0,C 180,E1 -6012.033,E2 -6012.033} C_VEL
LIN {X 0,Y 494.894,Z 528.017,A -85,B 0,C 180,E1 -6013.5,E2 -6013.5} C_VEL
LIN {X 0,Y 494.947,Z 529.452,A -85,B 0,C 180,E1 -6015.192,E2 -6015.192} C_VEL
LIN {X 0,Y 494.909,Z 529.466,A -85,B 0,C 180,E1 -6016.868,E2 -6016.868} C_VEL
LIN {X 0,Y 494.982,Z 528.075,A -85,B 0,C 180,E1 -6018.535,E2 -6018.535} C_VEL
LIN {X 0,Y 494.968,Z 525.31,A -85,B 0,C 180,E1 -6020.19,E2 -6020.19} C_VEL
LIN {X 0,Y 495.132,Z 521.095,A -85,B 0,C 180,E1 -6021.84,E2 -6021.84} C_VEL
LIN {X 0,Y 495.274,Z 515.342,A -85,B 0,C 180,E1 -6023.482,E2 -6023.482} C_VEL
LIN {X 0,Y 495.475,Z 508.881,A -85,B 0,C 180,E1 -6024.914,E2 -6024.914} C_VEL
LIN {X 0,Y 495.782,Z 500.899,A -85,B 0,C 180,E1 -6026.343,E2 -6026.343} C_VEL
LIN {X 0,Y 496.148,Z 492.567,A -85,B 0,C 180,E1 -6027.565,E2 -6027.565} C_VEL
LIN {X 0,Y 496.635,Z 482.558,A -85,B 0,C 180,E1 -6028.784,E2 -6028.784} C_VEL
LIN {X 0,Y 497.14,Z 471.401,A -85,B 0,C 180,E1 -6029.899,E2 -6029.899} C_VEL
LIN {X 0,Y 497.684,Z 460.331,A -85,B 0,C 180,E1 -6030.809,E2 -6030.809} C_VEL
LIN {X 0,Y 498.138,Z 448.344,A -85,B 0,C 180,E1 -6031.617,E2 -6031.617} C_VEL
LIN {X 0,Y 498.609,Z 435.073,A -85,B 0,C 180,E1 -6032.323,E2 -6032.323} C_VEL
LIN {X 0,Y 498.999,Z 421.233,A -85,B 0,C 180,E1 -6032.876,E2 -6032.876} C_VEL
LIN {X 0,Y 499.272,Z 406.689,A -85,B 0,C 180,E1 -6033.278,E2 -6033.278} C_VEL
LIN {X 0,Y 499.549,Z 379.538,A -85,B 0,C 180,E1 -6033.706,E2 -6033.706} C_VEL
LIN {X 0,Y 500.161,Z 282.451,A -85,B 0,C 180,E1 -6035.127,E2 -6035.127} C_VEL
LIN {X 0,Y 497.187,Z 268.345,A -85,B 0,C 180,E1 -6035.475,E2 -6035.475} C_VEL
LIN {X 0,Y 497.644,Z 255.719,A -85,B 0,C 180,E1 -6037.71,E2 -6037.71} C_VEL
LIN {X 0,Y 495.812,Z 246.352,A -85,B 0,C 180,E1 -6039.536,E2 -6039.536} C_VEL
LIN {X 0,Y 495.839,Z 246.349,A -85,B 0,C 180,E1 -6042.275,E2 -6042.275} C_VEL
LIN {X 0,Y 495.794,Z 246.355,A -85,B 0,C 180,E1 -6045.624,E2 -6045.624} C_VEL
LIN {X 0,Y 495.792,Z 246.35,A -85,B 0,C 180,E1 -6048.248,E2 -6048.248} C_VEL
LIN {X 0,Y 495.76,Z 246.351,A -85,B 0,C 180,E1 -6050.757,E2 -6050.757} C_VEL
LIN {X 0,Y 495.742,Z 246.357,A -85,B 0,C 180,E1 -6053.387,E2 -6053.387} C_VEL
LIN {X 0,Y 495.787,Z 246.351,A -85,B 0,C 180,E1 -6056.068,E2 -6056.068} C_VEL
LIN {X 0,Y 495.766,Z 246.351,A -85,B 0,C 180,E1 -6058.815,E2 -6058.815} C_VEL
LIN {X 0,Y 495.746,Z 246.359,A -85,B 0,C 180,E1 -6061.727,E2 -6061.727} C_VEL
LIN {X 0,Y 495.763,Z 246.351,A -85,B 0,C 180,E1 -6064.696,E2 -6064.696} C_VEL
LIN {X 0,Y 495.719,Z 246.363,A -85,B 0,C 180,E1 -6067.562,E2 -6067.562} C_VEL
LIN {X 0,Y 495.787,Z 246.349,A -85,B 0,C 180,E1 -6070.054,E2 -6070.054} C_VEL
LIN {X 0,Y 495.751,Z 246.355,A -85,B 0,C 180,E1 -6072.879,E2 -6072.879} C_VEL
LIN {X 0,Y 495.723,Z 246.356,A -85,B 0,C 180,E1 -6076,E2 -6076} C_VEL
LIN {X 0,Y 495.758,Z 246.353,A -85,B 0,C 180,E1 -6078.705,E2 -6078.705} C_VEL
LIN {X 0,Y 495.75,Z 246.358,A -85,B 0,C 180,E1 -6081.41,E2 -6081.41} C_VEL
LIN {X 0,Y 495.745,Z 246.354,A -85,B 0,C 180,E1 -6084.464,E2 -6084.464} C_VEL
LIN {X 0,Y 495.756,Z 246.356,A -85,B 0,C 180,E1 -6087.407,E2 -6087.407} C_VEL
LIN {X 0,Y 495.769,Z 246.35,A -85,B 0,C 180,E1 -6090.256,E2 -6090.256} C_VEL
LIN {X 0,Y 495.821,Z 246.348,A -85,B 0,C 180,E1 -6093.249,E2 -6093.249} C_VEL
LIN {X 0,Y 495.74,Z 246.354,A -85,B 0,C 180,E1 -6095.726,E2 -6095.726} C_VEL
LIN {X 0,Y 495.732,Z 246.357,A -85,B 0,C 180,E1 -6098.372,E2 -6098.372} C_VEL
LIN {X 0,Y 495.774,Z 246.356,A -85,B 0,C 180,E1 -6100.973,E2 -6100.973} C_VEL
LIN {X 0,Y 495.77,Z 246.35,A -85,B 0,C 180,E1 -6103.531,E2 -6103.531} C_VEL
LIN {X 0,Y 495.787,Z 246.349,A -85,B 0,C 180,E1 -6106.057,E2 -6106.057} C_VEL
LIN {X 0,Y 495.841,Z 246.348,A -85,B 0,C 180,E1 -6108.556,E2 -6108.556} C_VEL
LIN {X 0,Y 495.863,Z 246.339,A -85,B 0,C 180,E1 -6111.853,E2 -6111.853} C_VEL
LIN {X 0,Y 495.895,Z 246.339,A -85,B 0,C 180,E1 -6114.308,E2 -6114.308} C_VEL
LIN {X 0,Y 495.985,Z 246.323,A -85,B 0,C 180,E1 -6117.565,E2 -6117.565} C_VEL
LIN {X 0,Y 495.989,Z 246.325,A -85,B 0,C 180,E1 -6120.001,E2 -6120.001} C_VEL
LIN {X 0,Y 495.986,Z 246.332,A -85,B 0,C 180,E1 -6122.437,E2 -6122.437} C_VEL
LIN {X 0,Y 495.889,Z 246.336,A -85,B 0,C 180,E1 -6125.695,E2 -6125.695} C_VEL
LIN {X 0,Y 495.866,Z 246.344,A -85,B 0,C 180,E1 -6128.149,E2 -6128.149} C_VEL
LIN {X 0,Y 495.845,Z 246.341,A -85,B 0,C 180,E1 -6131.446,E2 -6131.446} C_VEL
LIN {X 0,Y 495.784,Z 246.35,A -85,B 0,C 180,E1 -6134.784,E2 -6134.784} C_VEL
LIN {X 0,Y 495.781,Z 246.349,A -85,B 0,C 180,E1 -6137.32,E2 -6137.32} C_VEL
LIN {X 0,Y 495.767,Z 246.356,A -85,B 0,C 180,E1 -6139.891,E2 -6139.891} C_VEL
LIN {X 0,Y 495.756,Z 246.352,A -85,B 0,C 180,E1 -6142.862,E2 -6142.862} C_VEL
LIN {X 0,Y 495.787,Z 246.356,A -85,B 0,C 180,E1 -6146.069,E2 -6146.069} C_VEL
LIN {X 0,Y 495.775,Z 246.349,A -85,B 0,C 180,E1 -6148.815,E2 -6148.815} C_VEL
LIN {X 0,Y 495.756,Z 246.358,A -85,B 0,C 180,E1 -6151.727,E2 -6151.727} C_VEL
LIN {X 0,Y 495.773,Z 246.35,A -85,B 0,C 180,E1 -6154.696,E2 -6154.696} C_VEL
LIN {X 0,Y 495.729,Z 246.36,A -85,B 0,C 180,E1 -6157.562,E2 -6157.562} C_VEL
LIN {X 0,Y 495.764,Z 246.35,A -85,B 0,C 180,E1 -6160.701,E2 -6160.701} C_VEL
LIN {X 0,Y 495.732,Z 246.359,A -85,B 0,C 180,E1 -6164.002,E2 -6164.002} C_VEL
LIN {X 0,Y 495.725,Z 246.358,A -85,B 0,C 180,E1 -6167.118,E2 -6167.118} C_VEL
LIN {X 0,Y 495.758,Z 246.355,A -85,B 0,C 180,E1 -6169.954,E2 -6169.954} C_VEL
LIN {X 0,Y 495.727,Z 246.355,A -85,B 0,C 180,E1 -6172.554,E2 -6172.554} C_VEL
LIN {X 0,Y 495.778,Z 246.358,A -85,B 0,C 180,E1 -6175.458,E2 -6175.458} C_VEL
LIN {X 0,Y 495.757,Z 246.357,A -85,B 0,C 180,E1 -6178.365,E2 -6178.365} C_VEL
LIN {X 0,Y 495.789,Z 246.356,A -85,B 0,C 180,E1 -6181.508,E2 -6181.508} C_VEL
LIN {X 0,Y 495.83,Z 246.446,A -85,B 0,C 180,E1 -6183.182,E2 -6183.182} C_VEL
LIN {X 0,Y 498.389,Z 258.467,A -85,B 0,C 180,E1 -6185.196,E2 -6185.196} C_VEL
LIN {X 0,Y 498.094,Z 268.467,A -85,B 0,C 180,E1 -6186.73,E2 -6186.73} C_VEL
LIN {X 0,Y 497.304,Z 289.845,A -85,B 0,C 180,E1 -6189.959,E2 -6189.959} C_VEL
LIN {X 0,Y 497.215,Z 294.165,A -85,B 0,C 180,E1 -6190.579,E2 -6190.579} C_VEL
LIN {X 0,Y 500.152,Z 310.845,A -85,B 0,C 180,E1 -6190.942,E2 -6190.942} C_VEL
LIN {X 0,Y 499.262,Z 431.913,A -85,B 0,C 180,E1 -6192.727,E2 -6192.727} C_VEL
LIN {X 0,Y 498.884,Z 446.504,A -85,B 0,C 180,E1 -6193.107,E2 -6193.107} C_VEL
LIN {X 0,Y 498.551,Z 460.003,A -85,B 0,C 180,E1 -6193.624,E2 -6193.624} C_VEL
LIN {X 0,Y 497.992,Z 474.021,A -85,B 0,C 180,E1 -6194.342,E2 -6194.342} C_VEL
LIN {X 0,Y 497.467,Z 486.557,A -85,B 0,C 180,E1 -6195.164,E2 -6195.164} C_VEL
LIN {X 0,Y 496.89,Z 499.184,A -85,B 0,C 180,E1 -6196.192,E2 -6196.192} C_VEL
LIN {X 0,Y 496.4,Z 510.436,A -85,B 0,C 180,E1 -6197.324,E2 -6197.324} C_VEL
LIN {X 0,Y 495.979,Z 520.522,A -85,B 0,C 180,E1 -6198.558,E2 -6198.558} C_VEL
LIN {X 0,Y 495.615,Z 528.9,A -85,B 0,C 180,E1 -6199.79,E2 -6199.79} C_VEL
LIN {X 0,Y 495.359,Z 536.911,A -85,B 0,C 180,E1 -6201.227,E2 -6201.227} C_VEL
LIN {X 0,Y 495.175,Z 543.361,A -85,B 0,C 180,E1 -6202.661,E2 -6202.661} C_VEL
LIN {X 0,Y 495.106,Z 549.081,A -85,B 0,C 180,E1 -6204.297,E2 -6204.297} C_VEL
LIN {X 0,Y 495.009,Z 553.229,A -85,B 0,C 180,E1 -6205.929,E2 -6205.929} C_VEL
LIN {X 0,Y 494.997,Z 555.938,A -85,B 0,C 180,E1 -6207.559,E2 -6207.559} C_VEL
LIN {X 0,Y 494.909,Z 557.278,A -85,B 0,C 180,E1 -6209.186,E2 -6209.186} C_VEL
LIN {X 0,Y 494.909,Z 557.275,A -85,B 0,C 180,E1 -6210.814,E2 -6210.814} C_VEL
LIN {X 0,Y 494.997,Z 555.932,A -85,B 0,C 180,E1 -6212.441,E2 -6212.441} C_VEL
LIN {X 0,Y 495.009,Z 553.217,A -85,B 0,C 180,E1 -6214.071,E2 -6214.071} C_VEL
LIN {X 0,Y 495.109,Z 549.059,A -85,B 0,C 180,E1 -6215.702,E2 -6215.702} C_VEL
LIN {X 0,Y 495.175,Z 543.33,A -85,B 0,C 180,E1 -6217.339,E2 -6217.339} C_VEL
LIN {X 0,Y 495.359,Z 536.874,A -85,B 0,C 180,E1 -6218.773,E2 -6218.773} C_VEL
LIN {X 0,Y 495.614,Z 528.855,A -85,B 0,C 180,E1 -6220.21,E2 -6220.21} C_VEL
LIN {X 0,Y 495.991,Z 520.471,A -85,B 0,C 180,E1 -6221.442,E2 -6221.442} C_VEL
LIN {X 0,Y 496.402,Z 510.377,A -85,B 0,C 180,E1 -6222.676,E2 -6222.676} C_VEL
LIN {X 0,Y 496.88,Z 499.119,A -85,B 0,C 180,E1 -6223.808,E2 -6223.808} C_VEL
LIN {X 0,Y 497.406,Z 487.929,A -85,B 0,C 180,E1 -6224.733,E2 -6224.733} C_VEL
LIN {X 0,Y 497.879,Z 475.742,A -85,B 0,C 180,E1 -6225.557,E2 -6225.557} C_VEL
LIN {X 0,Y 498.418,Z 463.356,A -85,B 0,C 180,E1 -6226.222,E2 -6226.222} C_VEL
LIN {X 0,Y 498.791,Z 449.589,A -85,B 0,C 180,E1 -6226.789,E2 -6226.789} C_VEL
LIN {X 0,Y 499.179,Z 435.405,A -85,B 0,C 180,E1 -6227.197,E2 -6227.197} C_VEL
LIN {X 0,Y 499.394,Z 415.703,A -85,B 0,C 180,E1 -6227.532,E2 -6227.532} C_VEL
LIN {X 0,Y 500.102,Z 310.262,A -85,B 0,C 180,E1 -6229.077,E2 -6229.077} C_VEL
LIN {X 0,Y 497.217,Z 293.669,A -85,B 0,C 180,E1 -6229.467,E2 -6229.467} C_VEL
LIN {X 0,Y 497.923,Z 272.926,A -85,B 0,C 180,E1 -6232.62,E2 -6232.62} C_VEL
LIN {X 0,Y 498.498,Z 260.247,A -85,B 0,C 180,E1 -6234.575,E2 -6234.575} C_VEL
LIN {X 0,Y 497.558,Z 254.098,A -85,B 0,C 180,E1 -6235.601,E2 -6235.601} C_VEL
LIN {X 0,Y 495.822,Z 246.352,A -85,B 0,C 180,E1 -6236.973,E2 -6236.973} C_VEL
LIN {X 0,Y 495.765,Z 246.358,A -85,B 0,C 180,E1 -6240.146,E2 -6240.146} C_VEL
LIN {X 0,Y 495.793,Z 246.354,A -85,B 0,C 180,E1 -6243.243,E2 -6243.243} C_VEL
LIN {X 0,Y 495.719,Z 246.365,A -85,B 0,C 180,E1 -6246.087,E2 -6246.087} C_VEL
LIN {X 0,Y 495.762,Z 246.359,A -85,B 0,C 180,E1 -6248.767,E2 -6248.767} C_VEL
LIN {X 0,Y 495.776,Z 246.351,A -85,B 0,C 180,E1 -6251.778,E2 -6251.778} C_VEL
LIN {X 0,Y 495.747,Z 246.354,A -85,B 0,C 180,E1 -6255.138,E2 -6255.138} C_VEL
LIN {X 0,Y 495.755,Z 246.359,A -85,B 0,C 180,E1 -6258.218,E2 -6258.218} C_VEL
LIN {X 0,Y 495.747,Z 246.355,A -85,B 0,C 180,E1 -6261.407,E2 -6261.407} C_VEL
LIN {X 0,Y 495.753,Z 246.349,A -85,B 0,C 180,E1 -6264.462,E2 -6264.462} C_VEL
LIN {X 0,Y 495.765,Z 246.353,A -85,B 0,C 180,E1 -6267.405,E2 -6267.405} C_VEL
LIN {X 0,Y 495.776,Z 246.354,A -85,B 0,C 180,E1 -6270.253,E2 -6270.253} C_VEL
LIN {X 0,Y 495.818,Z 246.344,A -85,B 0,C 180,E1 -6273.25,E2 -6273.25} C_VEL
LIN {X 0,Y 495.746,Z 246.358,A -85,B 0,C 180,E1 -6275.724,E2 -6275.724} C_VEL
LIN {X 0,Y 495.736,Z 246.356,A -85,B 0,C 180,E1 -6278.37,E2 -6278.37} C_VEL
LIN {X 0,Y 495.778,Z 246.349,A -85,B 0,C 180,E1 -6280.97,E2 -6280.97} C_VEL
LIN {X 0,Y 495.774,Z 246.355,A -85,B 0,C 180,E1 -6283.529,E2 -6283.529} C_VEL
LIN {X 0,Y 495.786,Z 246.351,A -85,B 0,C 180,E1 -6286.055,E2 -6286.055} C_VEL
LIN {X 0,Y 495.847,Z 246.338,A -85,B 0,C 180,E1 -6288.554,E2 -6288.554} C_VEL
LIN {X 0,Y 495.865,Z 246.338,A -85,B 0,C 180,E1 -6291.851,E2 -6291.851} C_VEL
LIN {X 0,Y 495.888,Z 246.336,A -85,B 0,C 180,E1 -6294.305,E2 -6294.305} C_VEL
LIN {X 0,Y 495.984,Z 246.329,A -85,B 0,C 180,E1 -6297.563,E2 -6297.563} C_VEL
LIN {X 0,Y 495.986,Z 246.323,A -85,B 0,C 180,E1 -6299.999,E2 -6299.999} C_VEL
LIN {X 0,Y 495.983,Z 246.323,A -85,B 0,C 180,E1 -6302.435,E2 -6302.435} C_VEL
LIN {X 0,Y 495.886,Z 246.336,A -85,B 0,C 180,E1 -6305.692,E2 -6305.692} C_VEL
LIN {X 0,Y 495.862,Z 246.339,A -85,B 0,C 180,E1 -6308.147,E2 -6308.147} C_VEL
LIN {X 0,Y 495.843,Z 246.345,A -85,B 0,C 180,E1 -6311.444,E2 -6311.444} C_VEL
LIN {X 0,Y 495.777,Z 246.353,A -85,B 0,C 180,E1 -6314.782,E2 -6314.782} C_VEL
LIN {X 0,Y 495.774,Z 246.352,A -85,B 0,C 180,E1 -6317.318,E2 -6317.318} C_VEL
LIN {X 0,Y 495.765,Z 246.351,A -85,B 0,C 180,E1 -6319.889,E2 -6319.889} C_VEL
LIN {X 0,Y 495.751,Z 246.359,A -85,B 0,C 180,E1 -6322.861,E2 -6322.861} C_VEL
LIN {X 0,Y 495.777,Z 246.351,A -85,B 0,C 180,E1 -6326.067,E2 -6326.067} C_VEL
LIN {X 0,Y 495.766,Z 246.355,A -85,B 0,C 180,E1 -6328.813,E2 -6328.813} C_VEL
LIN {X 0,Y 495.742,Z 246.351,A -85,B 0,C 180,E1 -6331.725,E2 -6331.725} C_VEL
LIN {X 0,Y 495.76,Z 246.352,A -85,B 0,C 180,E1 -6334.694,E2 -6334.694} C_VEL
LIN {X 0,Y 495.717,Z 246.359,A -85,B 0,C 180,E1 -6337.561,E2 -6337.561} C_VEL
LIN {X 0,Y 495.765,Z 246.357,A -85,B 0,C 180,E1 -6340.698,E2 -6340.698} C_VEL
LIN {X 0,Y 495.719,Z 246.36,A -85,B 0,C 180,E1 -6343.695,E2 -6343.695} C_VEL
LIN {X 0,Y 495.719,Z 246.364,A -85,B 0,C 180,E1 -6346.304,E2 -6346.304} C_VEL
LIN {X 0,Y 495.764,Z 246.355,A -85,B 0,C 180,E1 -6349.301,E2 -6349.301} C_VEL
LIN {X 0,Y 495.767,Z 246.404,A -85,B 0,C 180,E1 -6352.486,E2 -6352.486} C_VEL
LIN {X 0,Y 497.681,Z 256.08,A -85,B 0,C 180,E1 -6354.374,E2 -6354.374} C_VEL
LIN {X 0,Y 497.274,Z 268.499,A -85,B 0,C 180,E1 -6356.597,E2 -6356.597} C_VEL
LIN {X 0,Y 499.333,Z 278.316,A -85,B 0,C 180,E1 -6356.85,E2 -6356.85} C_VEL
LIN {X 0,Y 499.696,Z 282.146,A -85,B 0,C 180,E1 -6356.922,E2 -6356.922} C_VEL
LIN {X 0,Y 498.931,Z 287.973,A -85,B 0,C 180,E1 -6356.978,E2 -6356.978} C_VEL
LIN {X 0,Y 494.237,Z 303.406,A -85,B 0,C 180,E1 -6357.014,E2 -6357.014} C_VEL
LIN {X 0,Y 493.451,Z 309.372,A -85,B 0,C 180,E1 -6357.072,E2 -6357.072} C_VEL
LIN {X 0,Y 492.604,Z 405.671,A -85,B 0,C 180,E1 -6358.525,E2 -6358.525} C_VEL
LIN {X 0,Y 492.285,Z 420.153,A -85,B 0,C 180,E1 -6358.916,E2 -6358.916} C_VEL
LIN {X 0,Y 491.868,Z 433.976,A -85,B 0,C 180,E1 -6359.461,E2 -6359.461} C_VEL
LIN {X 0,Y 491.411,Z 445.934,A -85,B 0,C 180,E1 -6360.082,E2 -6360.082} C_VEL
LIN {X 0,Y 490.831,Z 459.084,A -85,B 0,C 180,E1 -6360.948,E2 -6360.948} C_VEL
LIN {X 0,Y 490.28,Z 470.536,A -85,B 0,C 180,E1 -6361.885,E2 -6361.885} C_VEL
LIN {X 0,Y 489.758,Z 480.963,A -85,B 0,C 180,E1 -6362.918,E2 -6362.918} C_VEL
LIN {X 0,Y 489.362,Z 490.259,A -85,B 0,C 180,E1 -6364.023,E2 -6364.023} C_VEL
LIN {X 0,Y 488.915,Z 499.659,A -85,B 0,C 180,E1 -6365.364,E2 -6365.364} C_VEL
LIN {X 0,Y 488.564,Z 507.321,A -85,B 0,C 180,E1 -6366.694,E2 -6366.694} C_VEL
LIN {X 0,Y 488.294,Z 513.613,A -85,B 0,C 180,E1 -6368.025,E2 -6368.025} C_VEL
LIN {X 0,Y 488.117,Z 518.765,A -85,B 0,C 180,E1 -6369.366,E2 -6369.366} C_VEL
LIN {X 0,Y 488.04,Z 522.734,A -85,B 0,C 180,E1 -6370.658,E2 -6370.658} C_VEL
LIN {X 0,Y 487.869,Z 526.588,A -85,B 0,C 180,E1 -6372.392,E2 -6372.392} C_VEL
LIN {X 0,Y 487.787,Z 528.913,A -85,B 0,C 180,E1 -6374.113,E2 -6374.113} C_VEL
LIN {X 0,Y 487.836,Z 529.8,A -85,B 0,C 180,E1 -6375.824,E2 -6375.824} C_VEL
LIN {X 0,Y 487.828,Z 529.294,A -85,B 0,C 180,E1 -6377.52,E2 -6377.52} C_VEL
LIN {X 0,Y 487.911,Z 528.522,A -85,B 0,C 180,E1 -6378.366,E2 -6378.366} C_VEL
LIN {X 0,Y 487.89,Z 525.942,A -85,B 0,C 180,E1 -6380.046,E2 -6380.046} C_VEL
LIN {X 0,Y 488.025,Z 521.899,A -85,B 0,C 180,E1 -6381.72,E2 -6381.72} C_VEL
LIN {X 0,Y 488.204,Z 516.318,A -85,B 0,C 180,E1 -6383.387,E2 -6383.387} C_VEL
LIN {X 0,Y 488.403,Z 510.047,A -85,B 0,C 180,E1 -6384.84,E2 -6384.84} C_VEL
LIN {X 0,Y 488.727,Z 502.27,A -85,B 0,C 180,E1 -6386.29,E2 -6386.29} C_VEL
LIN {X 0,Y 489.093,Z 494.177,A -85,B 0,C 180,E1 -6387.529,E2 -6387.529} C_VEL
LIN {X 0,Y 489.6,Z 484.451,A -85,B 0,C 180,E1 -6388.766,E2 -6388.766} C_VEL
LIN {X 0,Y 490.131,Z 473.69,A -85,B 0,C 180,E1 -6389.897,E2 -6389.897} C_VEL
LIN {X 0,Y 490.74,Z 461.765,A -85,B 0,C 180,E1 -6390.923,E2 -6390.923} C_VEL
LIN {X 0,Y 491.244,Z 450.046,A -85,B 0,C 180,E1 -6391.742,E2 -6391.742} C_VEL
LIN {X 0,Y 491.723,Z 437.224,A -85,B 0,C 180,E1 -6392.458,E2 -6392.458} C_VEL
LIN {X 0,Y 492.175,Z 423.289,A -85,B 0,C 180,E1 -6393.044,E2 -6393.044} C_VEL
LIN {X 0,Y 492.432,Z 408.596,A -85,B 0,C 180,E1 -6393.477,E2 -6393.477} C_VEL
LIN {X 0,Y 492.697,Z 389.249,A -85,B 0,C 180,E1 -6393.808,E2 -6393.808} C_VEL
LIN {X 0,Y 493.544,Z 284.109,A -85,B 0,C 180,E1 -6395.362,E2 -6395.362} C_VEL
LIN {X 0,Y 490.31,Z 268.613,A -85,B 0,C 180,E1 -6395.733,E2 -6395.733} C_VEL
LIN {X 0,Y 490.689,Z 256.974,A -85,B 0,C 180,E1 -6397.82,E2 -6397.82} C_VEL
LIN {X 0,Y 488.755,Z 247.232,A -85,B 0,C 180,E1 -6399.727,E2 -6399.727} C_VEL
LIN {X 0,Y 488.771,Z 247.227,A -85,B 0,C 180,E1 -6402.455,E2 -6402.455} C_VEL
LIN {X 0,Y 488.749,Z 247.233,A -85,B 0,C 180,E1 -6405.855,E2 -6405.855} C_VEL
LIN {X 0,Y 488.741,Z 247.227,A -85,B 0,C 180,E1 -6408.442,E2 -6408.442} C_VEL
LIN {X 0,Y 488.694,Z 247.232,A -85,B 0,C 180,E1 -6411.071,E2 -6411.071} C_VEL
LIN {X 0,Y 488.684,Z 247.241,A -85,B 0,C 180,E1 -6413.745,E2 -6413.745} C_VEL
LIN {X 0,Y 488.785,Z 247.221,A -85,B 0,C 180,E1 -6416.946,E2 -6416.946} C_VEL
LIN {X 0,Y 488.705,Z 247.23,A -85,B 0,C 180,E1 -6420.365,E2 -6420.365} C_VEL
LIN {X 0,Y 488.722,Z 247.236,A -85,B 0,C 180,E1 -6423.485,E2 -6423.485} C_VEL
LIN {X 0,Y 488.675,Z 247.234,A -85,B 0,C 180,E1 -6426.356,E2 -6426.356} C_VEL
LIN {X 0,Y 488.736,Z 247.232,A -85,B 0,C 180,E1 -6429.25,E2 -6429.25} C_VEL
LIN {X 0,Y 488.72,Z 247.228,A -85,B 0,C 180,E1 -6432.521,E2 -6432.521} C_VEL
LIN {X 0,Y 488.698,Z 247.238,A -85,B 0,C 180,E1 -6435.199,E2 -6435.199} C_VEL
LIN {X 0,Y 488.72,Z 247.234,A -85,B 0,C 180,E1 -6437.48,E2 -6437.48} C_VEL
LIN {X 0,Y 488.735,Z 247.229,A -85,B 0,C 180,E1 -6440.751,E2 -6440.751} C_VEL
LIN {X 0,Y 488.673,Z 247.235,A -85,B 0,C 180,E1 -6443.869,E2 -6443.869} C_VEL
LIN {X 0,Y 488.726,Z 247.233,A -85,B 0,C 180,E1 -6446.878,E2 -6446.878} C_VEL
LIN {X 0,Y 488.721,Z 247.228,A -85,B 0,C 180,E1 -6449.782,E2 -6449.782} C_VEL
LIN {X 0,Y 488.787,Z 247.227,A -85,B 0,C 180,E1 -6453.056,E2 -6453.056} C_VEL
LIN {X 0,Y 488.681,Z 247.234,A -85,B 0,C 180,E1 -6456.255,E2 -6456.255} C_VEL
LIN {X 0,Y 488.734,Z 247.231,A -85,B 0,C 180,E1 -6459.177,E2 -6459.177} C_VEL
LIN {X 0,Y 488.748,Z 247.225,A -85,B 0,C 180,E1 -6461.629,E2 -6461.629} C_VEL
LIN {X 0,Y 488.751,Z 247.229,A -85,B 0,C 180,E1 -6465.001,E2 -6465.001} C_VEL
LIN {X 0,Y 488.795,Z 247.223,A -85,B 0,C 180,E1 -6468.389,E2 -6468.389} C_VEL
LIN {X 0,Y 488.808,Z 247.217,A -85,B 0,C 180,E1 -6471.735,E2 -6471.735} C_VEL
LIN {X 0,Y 488.853,Z 247.215,A -85,B 0,C 180,E1 -6474.225,E2 -6474.225} C_VEL
LIN {X 0,Y 488.953,Z 247.199,A -85,B 0,C 180,E1 -6477.53,E2 -6477.53} C_VEL
LIN {X 0,Y 488.947,Z 247.204,A -85,B 0,C 180,E1 -6480.825,E2 -6480.825} C_VEL
LIN {X 0,Y 488.953,Z 247.207,A -85,B 0,C 180,E1 -6482.472,E2 -6482.472} C_VEL
LIN {X 0,Y 488.848,Z 247.213,A -85,B 0,C 180,E1 -6485.777,E2 -6485.777} C_VEL
LIN {X 0,Y 488.811,Z 247.224,A -85,B 0,C 180,E1 -6488.267,E2 -6488.267} C_VEL
LIN {X 0,Y 488.798,Z 247.219,A -85,B 0,C 180,E1 -6491.614,E2 -6491.614} C_VEL
LIN {X 0,Y 488.756,Z 247.224,A -85,B 0,C 180,E1 -6495.001,E2 -6495.001} C_VEL
LIN {X 0,Y 488.749,Z 247.229,A -85,B 0,C 180,E1 -6498.443,E2 -6498.443} C_VEL
LIN {X 0,Y 488.701,Z 247.23,A -85,B 0,C 180,E1 -6501.072,E2 -6501.072} C_VEL
LIN {X 0,Y 488.688,Z 247.236,A -85,B 0,C 180,E1 -6503.747,E2 -6503.747} C_VEL
LIN {X 0,Y 488.788,Z 247.22,A -85,B 0,C 180,E1 -6506.945,E2 -6506.945} C_VEL
LIN {X 0,Y 488.715,Z 247.232,A -85,B 0,C 180,E1 -6510.366,E2 -6510.366} C_VEL
LIN {X 0,Y 488.733,Z 247.23,A -85,B 0,C 180,E1 -6513.486,E2 -6513.486} C_VEL
LIN {X 0,Y 488.686,Z 247.234,A -85,B 0,C 180,E1 -6516.357,E2 -6516.357} C_VEL
LIN {X 0,Y 488.699,Z 247.233,A -85,B 0,C 180,E1 -6519.255,E2 -6519.255} C_VEL
LIN {X 0,Y 488.705,Z 247.237,A -85,B 0,C 180,E1 -6521.601,E2 -6521.601} C_VEL
LIN {X 0,Y 488.711,Z 247.229,A -85,B 0,C 180,E1 -6524.802,E2 -6524.802} C_VEL
LIN {X 0,Y 488.691,Z 247.238,A -85,B 0,C 180,E1 -6527.475,E2 -6527.475} C_VEL
LIN {X 0,Y 488.733,Z 247.234,A -85,B 0,C 180,E1 -6529.678,E2 -6529.678} C_VEL
LIN {X 0,Y 488.679,Z 247.234,A -85,B 0,C 180,E1 -6532.842,E2 -6532.842} C_VEL
LIN {X 0,Y 488.731,Z 247.232,A -85,B 0,C 180,E1 -6535.888,E2 -6535.888} C_VEL
LIN {X 0,Y 488.694,Z 247.238,A -85,B 0,C 180,E1 -6538.821,E2 -6538.821} C_VEL
LIN {X 0,Y 488.746,Z 247.232,A -85,B 0,C 180,E1 -6541.672,E2 -6541.672} C_VEL
LIN {X 0,Y 488.808,Z 247.329,A -85,B 0,C 180,E1 -6542.961,E2 -6542.961} C_VEL
LIN {X 0,Y 491.426,Z 259.604,A -85,B 0,C 180,E1 -6545.047,E2 -6545.047} C_VEL
LIN {X 0,Y 491.347,Z 265.624,A -85,B 0,C 180,E1 -6545.988,E2 -6545.988} C_VEL
LIN {X 0,Y 490.54,Z 285.301,A -85,B 0,C 180,E1 -6549.012,E2 -6549.012} C_VEL
LIN {X 0,Y 490.283,Z 293.724,A -85,B 0,C 180,E1 -6550.295,E2 -6550.295} C_VEL
LIN {X 0,Y 493.446,Z 313.003,A -85,B 0,C 180,E1 -6550.716,E2 -6550.716} C_VEL
LIN {X 0,Y 492.479,Z 431.437,A -85,B 0,C 180,E1 -6552.481,E2 -6552.481} C_VEL
LIN {X 0,Y 492.081,Z 446.289,A -85,B 0,C 180,E1 -6552.871,E2 -6552.871} C_VEL
LIN {X 0,Y 491.741,Z 459.699,A -85,B 0,C 180,E1 -6553.391,E2 -6553.391} C_VEL
LIN {X 0,Y 491.182,Z 471.978,A -85,B 0,C 180,E1 -6554.012,E2 -6554.012} C_VEL
LIN {X 0,Y 490.623,Z 484.88,A -85,B 0,C 180,E1 -6554.846,E2 -6554.846} C_VEL
LIN {X 0,Y 490.024,Z 496.593,A -85,B 0,C 180,E1 -6555.782,E2 -6555.782} C_VEL
LIN {X 0,Y 489.477,Z 508.303,A -85,B 0,C 180,E1 -6556.93,E2 -6556.93} C_VEL
LIN {X 0,Y 489.082,Z 517.885,A -85,B 0,C 180,E1 -6558.069,E2 -6558.069} C_VEL
LIN {X 0,Y 488.677,Z 527.419,A -85,B 0,C 180,E1 -6559.434,E2 -6559.434} C_VEL
LIN {X 0,Y 488.328,Z 535.694,A -85,B 0,C 180,E1 -6560.891,E2 -6560.891} C_VEL
LIN {X 0,Y 488.148,Z 541.481,A -85,B 0,C 180,E1 -6562.139,E2 -6562.139} C_VEL
LIN {X 0,Y 488.037,Z 546.752,A -85,B 0,C 180,E1 -6563.537,E2 -6563.537} C_VEL
LIN {X 0,Y 487.96,Z 551.142,A -85,B 0,C 180,E1 -6565.043,E2 -6565.043} C_VEL
LIN {X 0,Y 487.956,Z 554.56,A -85,B 0,C 180,E1 -6566.697,E2 -6566.697} C_VEL
LIN {X 0,Y 487.889,Z 556.579,A -85,B 0,C 180,E1 -6568.349,E2 -6568.349} C_VEL
LIN {X 0,Y 487.818,Z 557.245,A -85,B 0,C 180,E1 -6570,E2 -6570} C_VEL
LIN {X 0,Y 487.888,Z 556.573,A -85,B 0,C 180,E1 -6571.651,E2 -6571.651} C_VEL
LIN {X 0,Y 487.956,Z 554.549,A -85,B 0,C 180,E1 -6573.303,E2 -6573.303} C_VEL
LIN {X 0,Y 487.96,Z 551.122,A -85,B 0,C 180,E1 -6574.957,E2 -6574.957} C_VEL
LIN {X 0,Y 488.042,Z 546.194,A -85,B 0,C 180,E1 -6576.615,E2 -6576.615} C_VEL
LIN {X 0,Y 488.223,Z 539.619,A -85,B 0,C 180,E1 -6578.276,E2 -6578.276} C_VEL
LIN {X 0,Y 488.45,Z 532.308,A -85,B 0,C 180,E1 -6579.733,E2 -6579.733} C_VEL
LIN {X 0,Y 488.871,Z 523.256,A -85,B 0,C 180,E1 -6581.19,E2 -6581.19} C_VEL
LIN {X 0,Y 489.235,Z 513.759,A -85,B 0,C 180,E1 -6582.443,E2 -6582.443} C_VEL
LIN {X 0,Y 489.771,Z 502.182,A -85,B 0,C 180,E1 -6583.695,E2 -6583.695} C_VEL
LIN {X 0,Y 490.357,Z 490.386,A -85,B 0,C 180,E1 -6584.738,E2 -6584.738} C_VEL
LIN {X 0,Y 490.966,Z 477.263,A -85,B 0,C 180,E1 -6585.675,E2 -6585.675} C_VEL
LIN {X 0,Y 491.534,Z 464.329,A -85,B 0,C 180,E1 -6586.402,E2 -6586.402} C_VEL
LIN {X 0,Y 491.961,Z 450.776,A -85,B 0,C 180,E1 -6586.986,E2 -6586.986} C_VEL
LIN {X 0,Y 492.404,Z 436.707,A -85,B 0,C 180,E1 -6587.411,E2 -6587.411} C_VEL
LIN {X 0,Y 492.609,Z 421.284,A -85,B 0,C 180,E1 -6587.701,E2 -6587.701} C_VEL
LIN {X 0,Y 493.446,Z 311.252,A -85,B 0,C 180,E1 -6589.337,E2 -6589.337} C_VEL
LIN {X 0,Y 490.305,Z 293.461,A -85,B 0,C 180,E1 -6589.765,E2 -6589.765} C_VEL
LIN {X 0,Y 491.195,Z 271.441,A -85,B 0,C 180,E1 -6593.17,E2 -6593.17} C_VEL
LIN {X 0,Y 491.555,Z 260.204,A -85,B 0,C 180,E1 -6594.946,E2 -6594.946} C_VEL
LIN {X 0,Y 488.774,Z 247.227,A -85,B 0,C 180,E1 -6597.261,E2 -6597.261} C_VEL
LIN {X 0,Y 488.71,Z 247.237,A -85,B 0,C 180,E1 -6600.362,E2 -6600.362} C_VEL
LIN {X 0,Y 488.734,Z 247.233,A -85,B 0,C 180,E1 -6603.483,E2 -6603.483} C_VEL
LIN {X 0,Y 488.681,Z 247.245,A -85,B 0,C 180,E1 -6606.353,E2 -6606.353} C_VEL
LIN {X 0,Y 488.699,Z 247.235,A -85,B 0,C 180,E1 -6609.253,E2 -6609.253} C_VEL
LIN {X 0,Y 488.734,Z 247.234,A -85,B 0,C 180,E1 -6612.52,E2 -6612.52} C_VEL
LIN {X 0,Y 488.71,Z 247.231,A -85,B 0,C 180,E1 -6615.197,E2 -6615.197} C_VEL
LIN {X 0,Y 488.705,Z 247.237,A -85,B 0,C 180,E1 -6618.399,E2 -6618.399} C_VEL
LIN {X 0,Y 488.701,Z 247.232,A -85,B 0,C 180,E1 -6620.946,E2 -6620.946} C_VEL
LIN {X 0,Y 488.681,Z 247.231,A -85,B 0,C 180,E1 -6623.867,E2 -6623.867} C_VEL
LIN {X 0,Y 488.735,Z 247.227,A -85,B 0,C 180,E1 -6626.876,E2 -6626.876} C_VEL
LIN {X 0,Y 488.729,Z 247.231,A -85,B 0,C 180,E1 -6629.78,E2 -6629.78} C_VEL
LIN {X 0,Y 488.786,Z 247.219,A -85,B 0,C 180,E1 -6633.055,E2 -6633.055} C_VEL
LIN {X 0,Y 488.687,Z 247.234,A -85,B 0,C 180,E1 -6636.253,E2 -6636.253} C_VEL
LIN {X 0,Y 488.739,Z 247.228,A -85,B 0,C 180,E1 -6639.175,E2 -6639.175} C_VEL
LIN {X 0,Y 488.728,Z 247.228,A -85,B 0,C 180,E1 -6642.422,E2 -6642.422} C_VEL
LIN {X 0,Y 488.754,Z 247.224,A -85,B 0,C 180,E1 -6644.998,E2 -6644.998} C_VEL
LIN {X 0,Y 488.8,Z 247.215,A -85,B 0,C 180,E1 -6648.386,E2 -6648.386} C_VEL
LIN {X 0,Y 488.81,Z 247.218,A -85,B 0,C 180,E1 -6651.732,E2 -6651.732} C_VEL
LIN {X 0,Y 488.847,Z 247.213,A -85,B 0,C 180,E1 -6654.223,E2 -6654.223} C_VEL
LIN {X 0,Y 488.952,Z 247.204,A -85,B 0,C 180,E1 -6657.528,E2 -6657.528} C_VEL
LIN {X 0,Y 488.958,Z 247.199,A -85,B 0,C 180,E1 -6659.999,E2 -6659.999} C_VEL
LIN {X 0,Y 488.951,Z 247.199,A -85,B 0,C 180,E1 -6662.47,E2 -6662.47} C_VEL
LIN {X 0,Y 488.845,Z 247.212,A -85,B 0,C 180,E1 -6665.775,E2 -6665.775} C_VEL
LIN {X 0,Y 488.806,Z 247.218,A -85,B 0,C 180,E1 -6668.265,E2 -6668.265} C_VEL
LIN {X 0,Y 488.796,Z 247.221,A -85,B 0,C 180,E1 -6671.611,E2 -6671.611} C_VEL
LIN {X 0,Y 488.749,Z 247.232,A -85,B 0,C 180,E1 -6674.999,E2 -6674.999} C_VEL
LIN {X 0,Y 488.742,Z 247.228,A -85,B 0,C 180,E1 -6678.441,E2 -6678.441} C_VEL
LIN {X 0,Y 488.728,Z 247.233,A -85,B 0,C 180,E1 -6681.068,E2 -6681.068} C_VEL
LIN {X 0,Y 488.687,Z 247.231,A -85,B 0,C 180,E1 -6683.744,E2 -6683.744} C_VEL
LIN {X 0,Y 488.778,Z 247.227,A -85,B 0,C 180,E1 -6686.943,E2 -6686.943} C_VEL
LIN {X 0,Y 488.719,Z 247.23,A -85,B 0,C 180,E1 -6690.218,E2 -6690.218} C_VEL
LIN {X 0,Y 488.72,Z 247.229,A -85,B 0,C 180,E1 -6693.484,E2 -6693.484} C_VEL
LIN {X 0,Y 488.673,Z 247.237,A -85,B 0,C 180,E1 -6696.355,E2 -6696.355} C_VEL
LIN {X 0,Y 488.728,Z 247.227,A -85,B 0,C 180,E1 -6699.25,E2 -6699.25} C_VEL
LIN {X 0,Y 488.716,Z 247.234,A -85,B 0,C 180,E1 -6702.521,E2 -6702.521} C_VEL
LIN {X 0,Y 488.696,Z 247.233,A -85,B 0,C 180,E1 -6705.198,E2 -6705.198} C_VEL
LIN {X 0,Y 488.72,Z 247.232,A -85,B 0,C 180,E1 -6707.479,E2 -6707.479} C_VEL
LIN {X 0,Y 488.727,Z 247.235,A -85,B 0,C 180,E1 -6710.749,E2 -6710.749} C_VEL
LIN {X 0,Y 488.706,Z 247.316,A -85,B 0,C 180,E1 -6712.238,E2 -6712.238} C_VEL
LIN {X 0,Y 490.768,Z 257.388,A -85,B 0,C 180,E1 -6714.24,E2 -6714.24} C_VEL
LIN {X 0,Y 490.463,Z 269.014,A -85,B 0,C 180,E1 -6716.324,E2 -6716.324} C_VEL
LIN {X 0,Y 493.593,Z 283.671,A -85,B 0,C 180,E1 -6716.686,E2 -6716.686} C_VEL
LIN {X 0,Y 493.451,Z 309.372,A -85,B 0,C 180,E1 -6717.072,E2 -6717.072} C_VEL
LIN {X 0,Y 492.772,Z 315.217,A -85,B 0,C 180,E1 -6717.132,E2 -6717.132} C_VEL
LIN {X 0,Y 487.215,Z 334.251,A -85,B 0,C 180,E1 -6717.189,E2 -6717.189} C_VEL
LIN {X 0,Y 486.521,Z 340.097,A -85,B 0,C 180,E1 -6717.25,E2 -6717.25} C_VEL
LIN {X 0,Y 485.898,Z 405.625,A -85,B 0,C 180,E1 -6718.257,E2 -6718.257} C_VEL
LIN {X 0,Y 485.555,Z 419.925,A -85,B 0,C 180,E1 -6718.643,E2 -6718.643} C_VEL
LIN {X 0,Y 485.164,Z 433.377,A -85,B 0,C 180,E1 -6719.175,E2 -6719.175} C_VEL
LIN {X 0,Y 484.609,Z 446.445,A -85,B 0,C 180,E1 -6719.859,E2 -6719.859} C_VEL
LIN {X 0,Y 483.998,Z 459.253,A -85,B 0,C 180,E1 -6720.716,E2 -6720.716} C_VEL
LIN {X 0,Y 483.391,Z 470.907,A -85,B 0,C 180,E1 -6721.685,E2 -6721.685} C_VEL
LIN {X 0,Y 482.792,Z 482.24,A -85,B 0,C 180,E1 -6722.836,E2 -6722.836} C_VEL
LIN {X 0,Y 482.326,Z 492.29,A -85,B 0,C 180,E1 -6724.08,E2 -6724.08} C_VEL
LIN {X 0,Y 481.834,Z 501.336,A -85,B 0,C 180,E1 -6725.437,E2 -6725.437} C_VEL
LIN {X 0,Y 481.466,Z 509.109,A -85,B 0,C 180,E1 -6726.865,E2 -6726.865} C_VEL
LIN {X 0,Y 481.212,Z 514.805,A -85,B 0,C 180,E1 -6728.136,E2 -6728.136} C_VEL
LIN {X 0,Y 481.032,Z 519.669,A -85,B 0,C 180,E1 -6729.474,E2 -6729.474} C_VEL
LIN {X 0,Y 480.942,Z 523.509,A -85,B 0,C 180,E1 -6730.805,E2 -6730.805} C_VEL
LIN {X 0,Y 480.821,Z 526.426,A -85,B 0,C 180,E1 -6732.125,E2 -6732.125} C_VEL
LIN {X 0,Y 480.697,Z 528.915,A -85,B 0,C 180,E1 -6733.872,E2 -6733.872} C_VEL
LIN {X 0,Y 480.773,Z 529.614,A -85,B 0,C 180,E1 -6734.745,E2 -6734.745} C_VEL
LIN {X 0,Y 480.707,Z 529.959,A -85,B 0,C 180,E1 -6736.472,E2 -6736.472} C_VEL
LIN {X 0,Y 480.825,Z 528.799,A -85,B 0,C 180,E1 -6738.315,E2 -6738.315} C_VEL
LIN {X 0,Y 480.788,Z 526.509,A -85,B 0,C 180,E1 -6739.898,E2 -6739.898} C_VEL
LIN {X 0,Y 480.941,Z 522.678,A -85,B 0,C 180,E1 -6741.598,E2 -6741.598} C_VEL
LIN {X 0,Y 481.068,Z 518.768,A -85,B 0,C 180,E1 -6742.867,E2 -6742.867} C_VEL
LIN {X 0,Y 481.223,Z 513.967,A -85,B 0,C 180,E1 -6744.133,E2 -6744.133} C_VEL
LIN {X 0,Y 481.526,Z 507.056,A -85,B 0,C 180,E1 -6745.606,E2 -6745.606} C_VEL
LIN {X 0,Y 481.885,Z 498.537,A -85,B 0,C 180,E1 -6747.074,E2 -6747.074} C_VEL
LIN {X 0,Y 482.361,Z 489.65,A -85,B 0,C 180,E1 -6748.33,E2 -6748.33} C_VEL
LIN {X 0,Y 482.933,Z 478.932,A -85,B 0,C 180,E1 -6749.583,E2 -6749.583} C_VEL
LIN {X 0,Y 483.529,Z 468.071,A -85,B 0,C 180,E1 -6750.625,E2 -6750.625} C_VEL
LIN {X 0,Y 484.119,Z 456.195,A -85,B 0,C 180,E1 -6751.56,E2 -6751.56} C_VEL
LIN {X 0,Y 484.703,Z 442.98,A -85,B 0,C 180,E1 -6752.389,E2 -6752.389} C_VEL
LIN {X 0,Y 485.131,Z 430.3,A -85,B 0,C 180,E1 -6753.01,E2 -6753.01} C_VEL
LIN {X 0,Y 485.543,Z 415.875,A -85,B 0,C 180,E1 -6753.527,E2 -6753.527} C_VEL
LIN {X 0,Y 485.811,Z 401.54,A -85,B 0,C 180,E1 -6753.862,E2 -6753.862} C_VEL
LIN {X 0,Y 486.809,Z 284.857,A -85,B 0,C 180,E1 -6755.618,E2 -6755.618} C_VEL
LIN {X 0,Y 483.435,Z 268.72,A -85,B 0,C 180,E1 -6756.024,E2 -6756.024} C_VEL
LIN {X 0,Y 483.715,Z 258.228,A -85,B 0,C 180,E1 -6757.934,E2 -6757.934} C_VEL
LIN {X 0,Y 481.733,Z 248.106,A -85,B 0,C 180,E1 -6759.923,E2 -6759.923} C_VEL
LIN {X 0,Y 481.731,Z 248.103,A -85,B 0,C 180,E1 -6762.64,E2 -6762.64} C_VEL
LIN {X 0,Y 481.684,Z 248.109,A -85,B 0,C 180,E1 -6766.094,E2 -6766.094} C_VEL
LIN {X 0,Y 481.698,Z 248.103,A -85,B 0,C 180,E1 -6768.722,E2 -6768.722} C_VEL
LIN {X 0,Y 481.634,Z 248.115,A -85,B 0,C 180,E1 -6771.395,E2 -6771.395} C_VEL
LIN {X 0,Y 481.667,Z 248.11,A -85,B 0,C 180,E1 -6774.113,E2 -6774.113} C_VEL
LIN {X 0,Y 481.738,Z 248.1,A -85,B 0,C 180,E1 -6777.141,E2 -6777.141} C_VEL
LIN {X 0,Y 481.674,Z 248.112,A -85,B 0,C 180,E1 -6779.741,E2 -6779.741} C_VEL
LIN {X 0,Y 481.659,Z 248.108,A -85,B 0,C 180,E1 -6782.674,E2 -6782.674} C_VEL
LIN {X 0,Y 481.629,Z 248.117,A -85,B 0,C 180,E1 -6785.709,E2 -6785.709} C_VEL
LIN {X 0,Y 481.709,Z 248.109,A -85,B 0,C 180,E1 -6789.356,E2 -6789.356} C_VEL
LIN {X 0,Y 481.662,Z 248.108,A -85,B 0,C 180,E1 -6792.158,E2 -6792.158} C_VEL
LIN {X 0,Y 481.646,Z 248.109,A -85,B 0,C 180,E1 -6794.458,E2 -6794.458} C_VEL
LIN {X 0,Y 481.675,Z 248.108,A -85,B 0,C 180,E1 -6796.846,E2 -6796.846} C_VEL
LIN {X 0,Y 481.679,Z 248.105,A -85,B 0,C 180,E1 -6800.062,E2 -6800.062} C_VEL
LIN {X 0,Y 481.617,Z 248.12,A -85,B 0,C 180,E1 -6803.254,E2 -6803.254} C_VEL
LIN {X 0,Y 481.696,Z 248.103,A -85,B 0,C 180,E1 -6806.331,E2 -6806.331} C_VEL
LIN {X 0,Y 481.646,Z 248.113,A -85,B 0,C 180,E1 -6809.416,E2 -6809.416} C_VEL
LIN {X 0,Y 481.69,Z 248.104,A -85,B 0,C 180,E1 -6812.169,E2 -6812.169} C_VEL
LIN {X 0,Y 481.706,Z 248.11,A -85,B 0,C 180,E1 -6814.971,E2 -6814.971} C_VEL
LIN {X 0,Y 481.641,Z 248.11,A -85,B 0,C 180,E1 -6817.706,E2 -6817.706} C_VEL
LIN {X 0,Y 481.697,Z 248.106,A -85,B 0,C 180,E1 -6820.394,E2 -6820.394} C_VEL
LIN {X 0,Y 481.681,Z 248.11,A -85,B 0,C 180,E1 -6823.035,E2 -6823.035} C_VEL
LIN {X 0,Y 481.681,Z 248.105,A -85,B 0,C 180,E1 -6825.64,E2 -6825.64} C_VEL
LIN {X 0,Y 481.74,Z 248.1,A -85,B 0,C 180,E1 -6828.216,E2 -6828.216} C_VEL
LIN {X 0,Y 481.753,Z 248.096,A -85,B 0,C 180,E1 -6831.613,E2 -6831.613} C_VEL
LIN {X 0,Y 481.812,Z 248.091,A -85,B 0,C 180,E1 -6834.141,E2 -6834.141} C_VEL
LIN {X 0,Y 481.92,Z 248.075,A -85,B 0,C 180,E1 -6837.494,E2 -6837.494} C_VEL
LIN {X 0,Y 481.898,Z 248.081,A -85,B 0,C 180,E1 -6840.837,E2 -6840.837} C_VEL
LIN {X 0,Y 481.92,Z 248.083,A -85,B 0,C 180,E1 -6842.509,E2 -6842.509} C_VEL
LIN {X 0,Y 481.809,Z 248.091,A -85,B 0,C 180,E1 -6845.862,E2 -6845.862} C_VEL
LIN {X 0,Y 481.756,Z 248.103,A -85,B 0,C 180,E1 -6848.389,E2 -6848.389} C_VEL
LIN {X 0,Y 481.744,Z 248.099,A -85,B 0,C 180,E1 -6851.786,E2 -6851.786} C_VEL
LIN {X 0,Y 481.736,Z 248.098,A -85,B 0,C 180,E1 -6855.225,E2 -6855.225} C_VEL
LIN {X 0,Y 481.707,Z 248.103,A -85,B 0,C 180,E1 -6858.723,E2 -6858.723} C_VEL
LIN {X 0,Y 481.64,Z 248.111,A -85,B 0,C 180,E1 -6861.396,E2 -6861.396} C_VEL
LIN {X 0,Y 481.672,Z 248.114,A -85,B 0,C 180,E1 -6864.114,E2 -6864.114} C_VEL
LIN {X 0,Y 481.743,Z 248.097,A -85,B 0,C 180,E1 -6867.14,E2 -6867.14} C_VEL
LIN {X 0,Y 481.684,Z 248.11,A -85,B 0,C 180,E1 -6869.742,E2 -6869.742} C_VEL
LIN {X 0,Y 481.67,Z 248.107,A -85,B 0,C 180,E1 -6872.675,E2 -6872.675} C_VEL
LIN {X 0,Y 481.64,Z 248.117,A -85,B 0,C 180,E1 -6875.71,E2 -6875.71} C_VEL
LIN {X 0,Y 481.669,Z 248.106,A -85,B 0,C 180,E1 -6878.86,E2 -6878.86} C_VEL
LIN {X 0,Y 481.651,Z 248.114,A -85,B 0,C 180,E1 -6881.914,E2 -6881.914} C_VEL
LIN {X 0,Y 481.658,Z 248.108,A -85,B 0,C 180,E1 -6884.458,E2 -6884.458} C_VEL
LIN {X 0,Y 481.647,Z 248.114,A -85,B 0,C 180,E1 -6887.84,E2 -6887.84} C_VEL
LIN {X 0,Y 481.66,Z 248.108,A -85,B 0,C 180,E1 -6890.655,E2 -6890.655} C_VEL
LIN {X 0,Y 481.627,Z 248.118,A -85,B 0,C 180,E1 -6893.377,E2 -6893.377} C_VEL
LIN {X 0,Y 481.711,Z 248.101,A -85,B 0,C 180,E1 -6896.331,E2 -6896.331} C_VEL
LIN {X 0,Y 481.652,Z 248.119,A -85,B 0,C 180,E1 -6899.418,E2 -6899.418} C_VEL
LIN {X 0,Y 481.714,Z 248.107,A -85,B 0,C 180,E1 -6902.558,E2 -6902.558} C_VEL
LIN {X 0,Y 481.776,Z 248.344,A -85,B 0,C 180,E1 -6902.755,E2 -6902.755} C_VEL
LIN {X 0,Y 484.462,Z 260.8,A -85,B 0,C 180,E1 -6904.906,E2 -6904.906} C_VEL
LIN {X 0,Y 484.58,Z 265.024,A -85,B 0,C 180,E1 -6905.585,E2 -6905.585} C_VEL
LIN {X 0,Y 483.589,Z 286.446,A -85,B 0,C 180,E1 -6908.919,E2 -6908.919} C_VEL
LIN {X 0,Y 483.322,Z 293.509,A -85,B 0,C 180,E1 -6910.01,E2 -6910.01} C_VEL
LIN {X 0,Y 486.709,Z 313.696,A -85,B 0,C 180,E1 -6910.463,E2 -6910.463} C_VEL
LIN {X 0,Y 485.673,Z 431.942,A -85,B 0,C 180,E1 -6912.255,E2 -6912.255} C_VEL
LIN {X 0,Y 485.248,Z 446.634,A -85,B 0,C 180,E1 -6912.652,E2 -6912.652} C_VEL
LIN {X 0,Y 484.88,Z 459.295,A -85,B 0,C 180,E1 -6913.149,E2 -6913.149} C_VEL
LIN {X 0,Y 484.32,Z 471.771,A -85,B 0,C 180,E1 -6913.788,E2 -6913.788} C_VEL
LIN {X 0,Y 483.713,Z 484.573,A -85,B 0,C 180,E1 -6914.624,E2 -6914.624} C_VEL
LIN {X 0,Y 483.108,Z 496.316,A -85,B 0,C 180,E1 -6915.574,E2 -6915.574} C_VEL
LIN {X 0,Y 482.508,Z 508.049,A -85,B 0,C 180,E1 -6916.738,E2 -6916.738} C_VEL
LIN {X 0,Y 482.073,Z 517.983,A -85,B 0,C 180,E1 -6917.937,E2 -6917.937} C_VEL
LIN {X 0,Y 481.645,Z 527.196,A -85,B 0,C 180,E1 -6919.278,E2 -6919.278} C_VEL
LIN {X 0,Y 481.287,Z 535.482,A -85,B 0,C 180,E1 -6920.757,E2 -6920.757} C_VEL
LIN {X 0,Y 481.078,Z 541.272,A -85,B 0,C 180,E1 -6922.023,E2 -6922.023} C_VEL
LIN {X 0,Y 480.931,Z 546.99,A -85,B 0,C 180,E1 -6923.571,E2 -6923.571} C_VEL
LIN {X 0,Y 480.89,Z 550.941,A -85,B 0,C 180,E1 -6924.969,E2 -6924.969} C_VEL
LIN {X 0,Y 480.862,Z 554.36,A -85,B 0,C 180,E1 -6926.648,E2 -6926.648} C_VEL
LIN {X 0,Y 480.79,Z 556.379,A -85,B 0,C 180,E1 -6928.325,E2 -6928.325} C_VEL
LIN {X 0,Y 480.742,Z 557.046,A -85,B 0,C 180,E1 -6930,E2 -6930} C_VEL
LIN {X 0,Y 480.79,Z 556.373,A -85,B 0,C 180,E1 -6931.675,E2 -6931.675} C_VEL
LIN {X 0,Y 480.862,Z 554.349,A -85,B 0,C 180,E1 -6933.351,E2 -6933.351} C_VEL
LIN {X 0,Y 480.89,Z 550.923,A -85,B 0,C 180,E1 -6935.03,E2 -6935.03} C_VEL
LIN {X 0,Y 480.962,Z 545.994,A -85,B 0,C 180,E1 -6936.713,E2 -6936.713} C_VEL
LIN {X 0,Y 481.139,Z 539.421,A -85,B 0,C 180,E1 -6938.399,E2 -6938.399} C_VEL
LIN {X 0,Y 481.383,Z 532.115,A -85,B 0,C 180,E1 -6939.877,E2 -6939.877} C_VEL
LIN {X 0,Y 481.866,Z 523.077,A -85,B 0,C 180,E1 -6941.355,E2 -6941.355} C_VEL
LIN {X 0,Y 482.259,Z 513.595,A -85,B 0,C 180,E1 -6942.626,E2 -6942.626} C_VEL
LIN {X 0,Y 482.824,Z 502.04,A -85,B 0,C 180,E1 -6943.896,E2 -6943.896} C_VEL
LIN {X 0,Y 483.474,Z 490.276,A -85,B 0,C 180,E1 -6944.952,E2 -6944.952} C_VEL
LIN {X 0,Y 484.116,Z 477.197,A -85,B 0,C 180,E1 -6945.903,E2 -6945.903} C_VEL
LIN {X 0,Y 484.688,Z 464.943,A -85,B 0,C 180,E1 -6946.607,E2 -6946.607} C_VEL
LIN {X 0,Y 485.187,Z 450.888,A -85,B 0,C 180,E1 -6947.23,E2 -6947.23} C_VEL
LIN {X 0,Y 485.644,Z 437.02,A -85,B 0,C 180,E1 -6947.662,E2 -6947.662} C_VEL
LIN {X 0,Y 485.871,Z 421.893,A -85,B 0,C 180,E1 -6947.955,E2 -6947.955} C_VEL
LIN {X 0,Y 486.796,Z 312.48,A -85,B 0,C 180,E1 -6949.603,E2 -6949.603} C_VEL
LIN {X 0,Y 483.399,Z 293.234,A -85,B 0,C 180,E1 -6950.079,E2 -6950.079} C_VEL
LIN {X 0,Y 484.326,Z 272.803,A -85,B 0,C 180,E1 -6953.292,E2 -6953.292} C_VEL
LIN {X 0,Y 484.789,Z 262.975,A -85,B 0,C 180,E1 -6954.86,E2 -6954.86} C_VEL
LIN {X 0,Y 483.189,Z 254.591,A -85,B 0,C 180,E1 -6956.335,E2 -6956.335} C_VEL
LIN {X 0,Y 481.713,Z 248.105,A -85,B 0,C 180,E1 -6957.546,E2 -6957.546} C_VEL
LIN {X 0,Y 481.646,Z 248.118,A -85,B 0,C 180,E1 -6960.71,E2 -6960.71} C_VEL
LIN {X 0,Y 481.697,Z 248.111,A -85,B 0,C 180,E1 -6963.732,E2 -6963.732} C_VEL
LIN {X 0,Y 481.624,Z 248.118,A -85,B 0,C 180,E1 -6966.746,E2 -6966.746} C_VEL
LIN {X 0,Y 481.675,Z 248.113,A -85,B 0,C 180,E1 -6969.939,E2 -6969.939} C_VEL
LIN {X 0,Y 481.682,Z 248.107,A -85,B 0,C 180,E1 -6973.294,E2 -6973.294} C_VEL
LIN {X 0,Y 481.636,Z 248.114,A -85,B 0,C 180,E1 -6976.699,E2 -6976.699} C_VEL
LIN {X 0,Y 481.674,Z 248.112,A -85,B 0,C 180,E1 -6980.058,E2 -6980.058} C_VEL
LIN {X 0,Y 481.625,Z 248.11,A -85,B 0,C 180,E1 -6983.252,E2 -6983.252} C_VEL
LIN {X 0,Y 481.705,Z 248.107,A -85,B 0,C 180,E1 -6986.329,E2 -6986.329} C_VEL
LIN {X 0,Y 481.653,Z 248.108,A -85,B 0,C 180,E1 -6989.415,E2 -6989.415} C_VEL
LIN {X 0,Y 481.695,Z 248.106,A -85,B 0,C 180,E1 -6992.167,E2 -6992.167} C_VEL
LIN {X 0,Y 481.712,Z 248.102,A -85,B 0,C 180,E1 -6994.969,E2 -6994.969} C_VEL
LIN {X 0,Y 481.644,Z 248.117,A -85,B 0,C 180,E1 -6997.704,E2 -6997.704} C_VEL
LIN {X 0,Y 481.699,Z 248.103,A -85,B 0,C 180,E1 -7000.392,E2 -7000.392} C_VEL
LIN {X 0,Y 481.685,Z 248.106,A -85,B 0,C 180,E1 -7003.033,E2 -7003.033} C_VEL
LIN {X 0,Y 481.683,Z 248.113,A -85,B 0,C 180,E1 -7005.638,E2 -7005.638} C_VEL
LIN {X 0,Y 481.744,Z 248.095,A -85,B 0,C 180,E1 -7008.214,E2 -7008.214} C_VEL
LIN {X 0,Y 481.755,Z 248.099,A -85,B 0,C 180,E1 -7011.611,E2 -7011.611} C_VEL
LIN {X 0,Y 481.808,Z 248.091,A -85,B 0,C 180,E1 -7014.138,E2 -7014.138} C_VEL
LIN {X 0,Y 481.919,Z 248.08,A -85,B 0,C 180,E1 -7017.491,E2 -7017.491} C_VEL
LIN {X 0,Y 481.929,Z 248.075,A -85,B 0,C 180,E1 -7019.999,E2 -7019.999} C_VEL
LIN {X 0,Y 481.918,Z 248.075,A -85,B 0,C 180,E1 -7022.506,E2 -7022.506} C_VEL
LIN {X 0,Y 481.806,Z 248.088,A -85,B 0,C 180,E1 -7025.859,E2 -7025.859} C_VEL
LIN {X 0,Y 481.752,Z 248.098,A -85,B 0,C 180,E1 -7028.387,E2 -7028.387} C_VEL
LIN {X 0,Y 481.741,Z 248.099,A -85,B 0,C 180,E1 -7031.784,E2 -7031.784} C_VEL
LIN {X 0,Y 481.73,Z 248.105,A -85,B 0,C 180,E1 -7035.223,E2 -7035.223} C_VEL
LIN {X 0,Y 481.699,Z 248.108,A -85,B 0,C 180,E1 -7038.721,E2 -7038.721} C_VEL
LIN {X 0,Y 481.659,Z 248.11,A -85,B 0,C 180,E1 -7041.393,E2 -7041.393} C_VEL
LIN {X 0,Y 481.668,Z 248.106,A -85,B 0,C 180,E1 -7044.112,E2 -7044.112} C_VEL
LIN {X 0,Y 481.733,Z 248.102,A -85,B 0,C 180,E1 -7047.138,E2 -7047.138} C_VEL
LIN {X 0,Y 481.674,Z 248.105,A -85,B 0,C 180,E1 -7049.74,E2 -7049.74} C_VEL
LIN {X 0,Y 481.657,Z 248.116,A -85,B 0,C 180,E1 -7052.673,E2 -7052.673} C_VEL
LIN {X 0,Y 481.627,Z 248.109,A -85,B 0,C 180,E1 -7055.708,E2 -7055.708} C_VEL
LIN {X 0,Y 481.7,Z 248.102,A -85,B 0,C 180,E1 -7059.353,E2 -7059.353} C_VEL
LIN {X 0,Y 481.658,Z 248.111,A -85,B 0,C 180,E1 -7062.157,E2 -7062.157} C_VEL
LIN {X 0,Y 481.645,Z 248.118,A -85,B 0,C 180,E1 -7064.457,E2 -7064.457} C_VEL
LIN {X 0,Y 481.674,Z 248.111,A -85,B 0,C 180,E1 -7066.845,E2 -7066.845} C_VEL
LIN {X 0,Y 481.673,Z 248.114,A -85,B 0,C 180,E1 -7070.06,E2 -7070.06} C_VEL
LIN {X 0,Y 481.674,Z 248.263,A -85,B 0,C 180,E1 -7071.987,E2 -7071.987} C_VEL
LIN {X 0,Y 483.932,Z 259.365,A -85,B 0,C 180,E1 -7074.231,E2 -7074.231} C_VEL
LIN {X 0,Y 483.585,Z 269.053,A -85,B 0,C 180,E1 -7076.011,E2 -7076.011} C_VEL
LIN {X 0,Y 486.926,Z 284.734,A -85,B 0,C 180,E1 -7076.409,E2 -7076.409} C_VEL
LIN {X 0,Y 486.521,Z 340.097,A -85,B 0,C 180,E1 -7077.25,E2 -7077.25} C_VEL
LIN {X 0,Y 485.819,Z 345.945,A -85,B 0,C 180,E1 -7077.31,E2 -7077.31} C_VEL
LIN {X 0,Y 480.219,Z 364.976,A -85,B 0,C 180,E1 -7077.364,E2 -7077.364} C_VEL
LIN {X 0,Y 479.562,Z 370.821,A -85,B 0,C 180,E1 -7077.428,E2 -7077.428} C_VEL
LIN {X 0,Y 479.17,Z 406.751,A -85,B 0,C 180,E1 -7078.006,E2 -7078.006} C_VEL
LIN {X 0,Y 478.796,Z 420.955,A -85,B 0,C 180,E1 -7078.405,E2 -7078.405} C_VEL
LIN {X 0,Y 478.362,Z 434.423,A -85,B 0,C 180,E1 -7078.956,E2 -7078.956} C_VEL
LIN {X 0,Y 477.796,Z 446.948,A -85,B 0,C 180,E1 -7079.628,E2 -7079.628} C_VEL
LIN {X 0,Y 477.158,Z 459.645,A -85,B 0,C 180,E1 -7080.493,E2 -7080.493} C_VEL
LIN {X 0,Y 476.535,Z 471.314,A -85,B 0,C 180,E1 -7081.48,E2 -7081.48} C_VEL
LIN {X 0,Y 475.888,Z 482.201,A -85,B 0,C 180,E1 -7082.601,E2 -7082.601} C_VEL
LIN {X 0,Y 475.353,Z 492.564,A -85,B 0,C 180,E1 -7083.899,E2 -7083.899} C_VEL
LIN {X 0,Y 474.853,Z 501.636,A -85,B 0,C 180,E1 -7085.285,E2 -7085.285} C_VEL
LIN {X 0,Y 474.44,Z 509.188,A -85,B 0,C 180,E1 -7086.692,E2 -7086.692} C_VEL
LIN {X 0,Y 474.133,Z 515.931,A -85,B 0,C 180,E1 -7088.25,E2 -7088.25} C_VEL
LIN {X 0,Y 473.955,Z 520.646,A -85,B 0,C 180,E1 -7089.607,E2 -7089.607} C_VEL
LIN {X 0,Y 473.849,Z 524.295,A -85,B 0,C 180,E1 -7090.956,E2 -7090.956} C_VEL
LIN {X 0,Y 473.667,Z 527.769,A -85,B 0,C 180,E1 -7092.738,E2 -7092.738} C_VEL
LIN {X 0,Y 473.665,Z 529.698,A -85,B 0,C 180,E1 -7094.51,E2 -7094.51} C_VEL
LIN {X 0,Y 473.608,Z 530.198,A -85,B 0,C 180,E1 -7096.266,E2 -7096.266} C_VEL
LIN {X 0,Y 473.692,Z 529.31,A -85,B 0,C 180,E1 -7098.012,E2 -7098.012} C_VEL
LIN {X 0,Y 473.699,Z 527.053,A -85,B 0,C 180,E1 -7099.745,E2 -7099.745} C_VEL
LIN {X 0,Y 473.842,Z 523.381,A -85,B 0,C 180,E1 -7101.471,E2 -7101.471} C_VEL
LIN {X 0,Y 474.009,Z 518.216,A -85,B 0,C 180,E1 -7103.188,E2 -7103.188} C_VEL
LIN {X 0,Y 474.176,Z 513.213,A -85,B 0,C 180,E1 -7104.472,E2 -7104.472} C_VEL
LIN {X 0,Y 474.525,Z 506.077,A -85,B 0,C 180,E1 -7105.966,E2 -7105.966} C_VEL
LIN {X 0,Y 474.911,Z 498.63,A -85,B 0,C 180,E1 -7107.243,E2 -7107.243} C_VEL
LIN {X 0,Y 475.389,Z 489.719,A -85,B 0,C 180,E1 -7108.518,E2 -7108.518} C_VEL
LIN {X 0,Y 475.988,Z 478.964,A -85,B 0,C 180,E1 -7109.789,E2 -7109.789} C_VEL
LIN {X 0,Y 476.65,Z 468.054,A -85,B 0,C 180,E1 -7110.845,E2 -7110.845} C_VEL
LIN {X 0,Y 477.262,Z 456.127,A -85,B 0,C 180,E1 -7111.793,E2 -7111.793} C_VEL
LIN {X 0,Y 477.89,Z 442.813,A -85,B 0,C 180,E1 -7112.634,E2 -7112.634} C_VEL
LIN {X 0,Y 478.334,Z 430.026,A -85,B 0,C 180,E1 -7113.264,E2 -7113.264} C_VEL
LIN {X 0,Y 478.737,Z 416.315,A -85,B 0,C 180,E1 -7113.761,E2 -7113.761} C_VEL
LIN {X 0,Y 479.018,Z 402.141,A -85,B 0,C 180,E1 -7114.102,E2 -7114.102} C_VEL
LIN {X 0,Y 480.042,Z 285.516,A -85,B 0,C 180,E1 -7115.882,E2 -7115.882} C_VEL
LIN {X 0,Y 476.562,Z 268.941,A -85,B 0,C 180,E1 -7116.3,E2 -7116.3} C_VEL
LIN {X 0,Y 476.742,Z 259.464,A -85,B 0,C 180,E1 -7118.05,E2 -7118.05} C_VEL
LIN {X 0,Y 474.674,Z 248.985,A -85,B 0,C 180,E1 -7120.126,E2 -7120.126} C_VEL
LIN {X 0,Y 474.67,Z 248.983,A -85,B 0,C 180,E1 -7122.832,E2 -7122.832} C_VEL
LIN {X 0,Y 474.666,Z 248.987,A -85,B 0,C 180,E1 -7125.768,E2 -7125.768} C_VEL
LIN {X 0,Y 474.652,Z 248.981,A -85,B 0,C 180,E1 -7129.01,E2 -7129.01} C_VEL
LIN {X 0,Y 474.577,Z 248.998,A -85,B 0,C 180,E1 -7131.729,E2 -7131.729} C_VEL
LIN {X 0,Y 474.648,Z 248.981,A -85,B 0,C 180,E1 -7134.493,E2 -7134.493} C_VEL
LIN {X 0,Y 474.685,Z 248.981,A -85,B 0,C 180,E1 -7137.339,E2 -7137.339} C_VEL
LIN {X 0,Y 474.596,Z 248.988,A -85,B 0,C 180,E1 -7140.812,E2 -7140.812} C_VEL
LIN {X 0,Y 474.624,Z 248.986,A -85,B 0,C 180,E1 -7143.984,E2 -7143.984} C_VEL
LIN {X 0,Y 474.562,Z 248.993,A -85,B 0,C 180,E1 -7146.901,E2 -7146.901} C_VEL
LIN {X 0,Y 474.653,Z 248.985,A -85,B 0,C 180,E1 -7149.654,E2 -7149.654} C_VEL
LIN {X 0,Y 474.639,Z 248.985,A -85,B 0,C 180,E1 -7152.93,E2 -7152.93} C_VEL
LIN {X 0,Y 474.604,Z 248.988,A -85,B 0,C 180,E1 -7155.897,E2 -7155.897} C_VEL
LIN {X 0,Y 474.633,Z 248.988,A -85,B 0,C 180,E1 -7159.039,E2 -7159.039} C_VEL
LIN {X 0,Y 474.606,Z 248.988,A -85,B 0,C 180,E1 -7161.703,E2 -7161.703} C_VEL
LIN {X 0,Y 474.617,Z 248.988,A -85,B 0,C 180,E1 -7164.727,E2 -7164.727} C_VEL
LIN {X 0,Y 474.624,Z 248.985,A -85,B 0,C 180,E1 -7167.789,E2 -7167.789} C_VEL
LIN {X 0,Y 474.62,Z 248.991,A -85,B 0,C 180,E1 -7170.883,E2 -7170.883} C_VEL
LIN {X 0,Y 474.654,Z 248.981,A -85,B 0,C 180,E1 -7173.63,E2 -7173.63} C_VEL
LIN {X 0,Y 474.624,Z 248.989,A -85,B 0,C 180,E1 -7176.642,E2 -7176.642} C_VEL
LIN {X 0,Y 474.645,Z 248.982,A -85,B 0,C 180,E1 -7180.091,E2 -7180.091} C_VEL
LIN {X 0,Y 474.641,Z 248.99,A -85,B 0,C 180,E1 -7182.776,E2 -7182.776} C_VEL
LIN {X 0,Y 474.638,Z 248.983,A -85,B 0,C 180,E1 -7185.422,E2 -7185.422} C_VEL
LIN {X 0,Y 474.694,Z 248.976,A -85,B 0,C 180,E1 -7188.039,E2 -7188.039} C_VEL
LIN {X 0,Y 474.719,Z 248.972,A -85,B 0,C 180,E1 -7191.488,E2 -7191.488} C_VEL
LIN {X 0,Y 474.774,Z 248.967,A -85,B 0,C 180,E1 -7194.054,E2 -7194.054} C_VEL
LIN {X 0,Y 474.886,Z 248.951,A -85,B 0,C 180,E1 -7197.457,E2 -7197.457} C_VEL
LIN {X 0,Y 474.903,Z 248.952,A -85,B 0,C 180,E1 -7200.001,E2 -7200.001} C_VEL
LIN {X 0,Y 474.887,Z 248.958,A -85,B 0,C 180,E1 -7202.546,E2 -7202.546} C_VEL
LIN {X 0,Y 474.772,Z 248.968,A -85,B 0,C 180,E1 -7205.949,E2 -7205.949} C_VEL
LIN {X 0,Y 474.721,Z 248.978,A -85,B 0,C 180,E1 -7208.515,E2 -7208.515} C_VEL
LIN {X 0,Y 474.697,Z 248.979,A -85,B 0,C 180,E1 -7211.964,E2 -7211.964} C_VEL
LIN {X 0,Y 474.696,Z 248.978,A -85,B 0,C 180,E1 -7215.778,E2 -7215.778} C_VEL
LIN {X 0,Y 474.659,Z 248.98,A -85,B 0,C 180,E1 -7219.011,E2 -7219.011} C_VEL
LIN {X 0,Y 474.584,Z 248.993,A -85,B 0,C 180,E1 -7221.73,E2 -7221.73} C_VEL
LIN {X 0,Y 474.654,Z 248.983,A -85,B 0,C 180,E1 -7224.494,E2 -7224.494} C_VEL
LIN {X 0,Y 474.677,Z 248.978,A -85,B 0,C 180,E1 -7227.336,E2 -7227.336} C_VEL
LIN {X 0,Y 474.61,Z 248.99,A -85,B 0,C 180,E1 -7230.231,E2 -7230.231} C_VEL
LIN {X 0,Y 474.64,Z 248.983,A -85,B 0,C 180,E1 -7233.221,E2 -7233.221} C_VEL
LIN {X 0,Y 474.591,Z 248.99,A -85,B 0,C 180,E1 -7236.324,E2 -7236.324} C_VEL
LIN {X 0,Y 474.626,Z 248.991,A -85,B 0,C 180,E1 -7239.649,E2 -7239.649} C_VEL
LIN {X 0,Y 474.613,Z 248.986,A -85,B 0,C 180,E1 -7242.935,E2 -7242.935} C_VEL
LIN {X 0,Y 474.609,Z 248.991,A -85,B 0,C 180,E1 -7245.896,E2 -7245.896} C_VEL
LIN {X 0,Y 474.627,Z 248.985,A -85,B 0,C 180,E1 -7249.042,E2 -7249.042} C_VEL
LIN {X 0,Y 474.609,Z 248.992,A -85,B 0,C 180,E1 -7251.705,E2 -7251.705} C_VEL
LIN {X 0,Y 474.624,Z 248.984,A -85,B 0,C 180,E1 -7254.726,E2 -7254.726} C_VEL
LIN {X 0,Y 474.637,Z 248.992,A -85,B 0,C 180,E1 -7257.789,E2 -7257.789} C_VEL
LIN {X 0,Y 474.625,Z 248.991,A -85,B 0,C 180,E1 -7260.885,E2 -7260.885} C_VEL
LIN {X 0,Y 474.693,Z 249.037,A -85,B 0,C 180,E1 -7262.492,E2 -7262.492} C_VEL
LIN {X 0,Y 477.659,Z 263.262,A -85,B 0,C 180,E1 -7264.976,E2 -7264.976} C_VEL
LIN {X 0,Y 477.244,Z 274.704,A -85,B 0,C 180,E1 -7266.801,E2 -7266.801} C_VEL
LIN {X 0,Y 476.408,Z 293.408,A -85,B 0,C 180,E1 -7269.735,E2 -7269.735} C_VEL
LIN {X 0,Y 479.986,Z 314.366,A -85,B 0,C 180,E1 -7270.207,E2 -7270.207} C_VEL
LIN {X 0,Y 478.911,Z 431.117,A -85,B 0,C 180,E1 -7271.996,E2 -7271.996} C_VEL
LIN {X 0,Y 478.457,Z 446.028,A -85,B 0,C 180,E1 -7272.398,E2 -7272.398} C_VEL
LIN {X 0,Y 478.043,Z 458.793,A -85,B 0,C 180,E1 -7272.901,E2 -7272.901} C_VEL
LIN {X 0,Y 477.466,Z 471.56,A -85,B 0,C 180,E1 -7273.563,E2 -7273.563} C_VEL
LIN {X 0,Y 476.828,Z 484.189,A -85,B 0,C 180,E1 -7274.396,E2 -7274.396} C_VEL
LIN {X 0,Y 476.211,Z 495.979,A -85,B 0,C 180,E1 -7275.361,E2 -7275.361} C_VEL
LIN {X 0,Y 475.547,Z 507.748,A -85,B 0,C 180,E1 -7276.54,E2 -7276.54} C_VEL
LIN {X 0,Y 475.046,Z 518.403,A -85,B 0,C 180,E1 -7277.847,E2 -7277.847} C_VEL
LIN {X 0,Y 474.61,Z 526.946,A -85,B 0,C 180,E1 -7279.117,E2 -7279.117} C_VEL
LIN {X 0,Y 474.257,Z 535.25,A -85,B 0,C 180,E1 -7280.619,E2 -7280.619} C_VEL
LIN {X 0,Y 474.02,Z 541.047,A -85,B 0,C 180,E1 -7281.903,E2 -7281.903} C_VEL
LIN {X 0,Y 473.858,Z 547.088,A -85,B 0,C 180,E1 -7283.572,E2 -7283.572} C_VEL
LIN {X 0,Y 473.82,Z 550.732,A -85,B 0,C 180,E1 -7284.894,E2 -7284.894} C_VEL
LIN {X 0,Y 473.756,Z 554.154,A -85,B 0,C 180,E1 -7286.598,E2 -7286.598} C_VEL
LIN {X 0,Y 473.696,Z 556.177,A -85,B 0,C 180,E1 -7288.3,E2 -7288.3} C_VEL
LIN {X 0,Y 473.668,Z 556.847,A -85,B 0,C 180,E1 -7290,E2 -7290} C_VEL
LIN {X 0,Y 473.696,Z 556.176,A -85,B 0,C 180,E1 -7291.7,E2 -7291.7} C_VEL
LIN {X 0,Y 473.756,Z 554.153,A -85,B 0,C 180,E1 -7293.402,E2 -7293.402} C_VEL
LIN {X 0,Y 473.82,Z 550.731,A -85,B 0,C 180,E1 -7295.106,E2 -7295.106} C_VEL
LIN {X 0,Y 473.892,Z 545.808,A -85,B 0,C 180,E1 -7296.814,E2 -7296.814} C_VEL
LIN {X 0,Y 474.074,Z 539.242,A -85,B 0,C 180,E1 -7298.525,E2 -7298.525} C_VEL
LIN {X 0,Y 474.337,Z 531.95,A -85,B 0,C 180,E1 -7300.026,E2 -7300.026} C_VEL
LIN {X 0,Y 474.86,Z 522.935,A -85,B 0,C 180,E1 -7301.525,E2 -7301.525} C_VEL
LIN {X 0,Y 475.291,Z 513.481,A -85,B 0,C 180,E1 -7302.814,E2 -7302.814} C_VEL
LIN {X 0,Y 475.835,Z 503.028,A -85,B 0,C 180,E1 -7303.996,E2 -7303.996} C_VEL
LIN {X 0,Y 476.512,Z 491.51,A -85,B 0,C 180,E1 -7305.067,E2 -7305.067} C_VEL
LIN {X 0,Y 477.183,Z 478.753,A -85,B 0,C 180,E1 -7306.03,E2 -7306.03} C_VEL
LIN {X 0,Y 477.844,Z 465.581,A -85,B 0,C 180,E1 -7306.817,E2 -7306.817} C_VEL
LIN {X 0,Y 478.358,Z 452.171,A -85,B 0,C 180,E1 -7307.434,E2 -7307.434} C_VEL
LIN {X 0,Y 478.873,Z 438.378,A -85,B 0,C 180,E1 -7307.889,E2 -7307.889} C_VEL
LIN {X 0,Y 479.184,Z 424.289,A -85,B 0,C 180,E1 -7308.187,E2 -7308.187} C_VEL
LIN {X 0,Y 480.179,Z 313.53,A -85,B 0,C 180,E1 -7309.884,E2 -7309.884} C_VEL
LIN {X 0,Y 476.508,Z 293.162,A -85,B 0,C 180,E1 -7310.383,E2 -7310.383} C_VEL
LIN {X 0,Y 477.588,Z 271.762,A -85,B 0,C 180,E1 -7313.803,E2 -7313.803} C_VEL
LIN {X 0,Y 477.93,Z 264.377,A -85,B 0,C 180,E1 -7315.009,E2 -7315.009} C_VEL
LIN {X 0,Y 475.666,Z 253.231,A -85,B 0,C 180,E1 -7317.021,E2 -7317.021} C_VEL
LIN {X 0,Y 474.664,Z 248.984,A -85,B 0,C 180,E1 -7317.859,E2 -7317.859} C_VEL
LIN {X 0,Y 474.599,Z 248.994,A -85,B 0,C 180,E1 -7321.217,E2 -7321.217} C_VEL
LIN {X 0,Y 474.631,Z 248.993,A -85,B 0,C 180,E1 -7324.24,E2 -7324.24} C_VEL
LIN {X 0,Y 474.589,Z 248.99,A -85,B 0,C 180,E1 -7327.383,E2 -7327.383} C_VEL
LIN {X 0,Y 474.626,Z 248.99,A -85,B 0,C 180,E1 -7329.646,E2 -7329.646} C_VEL
LIN {X 0,Y 474.651,Z 248.984,A -85,B 0,C 180,E1 -7332.929,E2 -7332.929} C_VEL
LIN {X 0,Y 474.607,Z 248.991,A -85,B 0,C 180,E1 -7335.894,E2 -7335.894} C_VEL
LIN {X 0,Y 474.625,Z 248.986,A -85,B 0,C 180,E1 -7339.04,E2 -7339.04} C_VEL
LIN {X 0,Y 474.607,Z 248.991,A -85,B 0,C 180,E1 -7341.703,E2 -7341.703} C_VEL
LIN {X 0,Y 474.626,Z 248.978,A -85,B 0,C 180,E1 -7344.725,E2 -7344.725} C_VEL
LIN {X 0,Y 474.634,Z 248.989,A -85,B 0,C 180,E1 -7347.787,E2 -7347.787} C_VEL
LIN {X 0,Y 474.626,Z 248.985,A -85,B 0,C 180,E1 -7350.882,E2 -7350.882} C_VEL
LIN {X 0,Y 474.655,Z 248.984,A -85,B 0,C 180,E1 -7353.627,E2 -7353.627} C_VEL
LIN {X 0,Y 474.63,Z 248.983,A -85,B 0,C 180,E1 -7356.64,E2 -7356.64} C_VEL
LIN {X 0,Y 474.648,Z 248.984,A -85,B 0,C 180,E1 -7360.088,E2 -7360.088} C_VEL
LIN {X 0,Y 474.644,Z 248.982,A -85,B 0,C 180,E1 -7362.773,E2 -7362.773} C_VEL
LIN {X 0,Y 474.641,Z 248.986,A -85,B 0,C 180,E1 -7365.42,E2 -7365.42} C_VEL
LIN {X 0,Y 474.697,Z 248.974,A -85,B 0,C 180,E1 -7368.036,E2 -7368.036} C_VEL
LIN {X 0,Y 474.721,Z 248.977,A -85,B 0,C 180,E1 -7371.485,E2 -7371.485} C_VEL
LIN {X 0,Y 474.771,Z 248.968,A -85,B 0,C 180,E1 -7374.051,E2 -7374.051} C_VEL
LIN {X 0,Y 474.885,Z 248.955,A -85,B 0,C 180,E1 -7377.454,E2 -7377.454} C_VEL
LIN {X 0,Y 474.867,Z 248.956,A -85,B 0,C 180,E1 -7380.847,E2 -7380.847} C_VEL
LIN {X 0,Y 474.885,Z 248.952,A -85,B 0,C 180,E1 -7382.543,E2 -7382.543} C_VEL
LIN {X 0,Y 474.768,Z 248.965,A -85,B 0,C 180,E1 -7385.946,E2 -7385.946} C_VEL
LIN {X 0,Y 474.717,Z 248.975,A -85,B 0,C 180,E1 -7388.512,E2 -7388.512} C_VEL
LIN {X 0,Y 474.694,Z 248.977,A -85,B 0,C 180,E1 -7391.961,E2 -7391.961} C_VEL
LIN {X 0,Y 474.687,Z 248.979,A -85,B 0,C 180,E1 -7395.455,E2 -7395.455} C_VEL
LIN {X 0,Y 474.653,Z 248.987,A -85,B 0,C 180,E1 -7399.009,E2 -7399.009} C_VEL
LIN {X 0,Y 474.596,Z 248.989,A -85,B 0,C 180,E1 -7401.727,E2 -7401.727} C_VEL
LIN {X 0,Y 474.648,Z 248.984,A -85,B 0,C 180,E1 -7404.492,E2 -7404.492} C_VEL
LIN {X 0,Y 474.667,Z 248.981,A -85,B 0,C 180,E1 -7407.334,E2 -7407.334} C_VEL
LIN {X 0,Y 474.599,Z 248.988,A -85,B 0,C 180,E1 -7410.229,E2 -7410.229} C_VEL
LIN {X 0,Y 474.628,Z 248.986,A -85,B 0,C 180,E1 -7413.219,E2 -7413.219} C_VEL
LIN {X 0,Y 474.578,Z 248.992,A -85,B 0,C 180,E1 -7416.323,E2 -7416.323} C_VEL
LIN {X 0,Y 474.636,Z 248.982,A -85,B 0,C 180,E1 -7419.65,E2 -7419.65} C_VEL
LIN {X 0,Y 474.636,Z 248.987,A -85,B 0,C 180,E1 -7422.93,E2 -7422.93} C_VEL
LIN {X 0,Y 474.603,Z 248.992,A -85,B 0,C 180,E1 -7425.896,E2 -7425.896} C_VEL
LIN {X 0,Y 474.63,Z 248.988,A -85,B 0,C 180,E1 -7429.038,E2 -7429.038} C_VEL
LIN {X 0,Y 474.639,Z 249.079,A -85,B 0,C 180,E1 -7431.697,E2 -7431.697} C_VEL
LIN {X 0,Y 477.056,Z 260.851,A -85,B 0,C 180,E1 -7434.118,E2 -7434.118} C_VEL
LIN {X 0,Y 476.719,Z 269.276,A -85,B 0,C 180,E1 -7435.686,E2 -7435.686} C_VEL
LIN {X 0,Y 480.276,Z 285.561,A -85,B 0,C 180,E1 -7436.116,E2 -7436.116} C_VEL
LIN {X 0,Y 479.975,Z 326.612,A -85,B 0,C 180,E1 -7436.75,E2 -7436.75} C_VEL
LIN {X 0,Y 479.562,Z 370.821,A -85,B 0,C 180,E1 -7437.428,E2 -7437.428} C_VEL
LIN {X 0,Y 478.88,Z 376.678,A -85,B 0,C 180,E1 -7437.488,E2 -7437.488} C_VEL
LIN {X 0,Y 473.196,Z 395.708,A -85,B 0,C 180,E1 -7437.537,E2 -7437.537} C_VEL
LIN {X 0,Y 472.595,Z 401.54,A -85,B 0,C 180,E1 -7437.615,E2 -7437.615} C_VEL
LIN {X 0,Y 472.25,Z 416.161,A -85,B 0,C 180,E1 -7437.964,E2 -7437.964} C_VEL
LIN {X 0,Y 471.841,Z 428.87,A -85,B 0,C 180,E1 -7438.424,E2 -7438.424} C_VEL
LIN {X 0,Y 471.234,Z 442.625,A -85,B 0,C 180,E1 -7439.097,E2 -7439.097} C_VEL
LIN {X 0,Y 470.628,Z 455.592,A -85,B 0,C 180,E1 -7439.925,E2 -7439.925} C_VEL
LIN {X 0,Y 469.885,Z 467.983,A -85,B 0,C 180,E1 -7440.916,E2 -7440.916} C_VEL
LIN {X 0,Y 469.141,Z 479.935,A -85,B 0,C 180,E1 -7442.107,E2 -7442.107} C_VEL
LIN {X 0,Y 468.58,Z 489.492,A -85,B 0,C 180,E1 -7443.26,E2 -7443.26} C_VEL
LIN {X 0,Y 468.035,Z 499.114,A -85,B 0,C 180,E1 -7444.663,E2 -7444.663} C_VEL
LIN {X 0,Y 467.569,Z 506.991,A -85,B 0,C 180,E1 -7446.057,E2 -7446.057} C_VEL
LIN {X 0,Y 467.214,Z 513.439,A -85,B 0,C 180,E1 -7447.445,E2 -7447.445} C_VEL
LIN {X 0,Y 466.957,Z 519.001,A -85,B 0,C 180,E1 -7448.924,E2 -7448.924} C_VEL
LIN {X 0,Y 466.786,Z 523.986,A -85,B 0,C 180,E1 -7450.657,E2 -7450.657} C_VEL
LIN {X 0,Y 466.6,Z 527.628,A -85,B 0,C 180,E1 -7452.468,E2 -7452.468} C_VEL
LIN {X 0,Y 466.567,Z 529.752,A -85,B 0,C 180,E1 -7454.269,E2 -7454.269} C_VEL
LIN {X 0,Y 466.514,Z 530.434,A -85,B 0,C 180,E1 -7456.053,E2 -7456.053} C_VEL
LIN {X 0,Y 466.579,Z 529.699,A -85,B 0,C 180,E1 -7457.826,E2 -7457.826} C_VEL
LIN {X 0,Y 466.621,Z 527.588,A -85,B 0,C 180,E1 -7459.588,E2 -7459.588} C_VEL
LIN {X 0,Y 466.758,Z 524.069,A -85,B 0,C 180,E1 -7461.34,E2 -7461.34} C_VEL
LIN {X 0,Y 466.914,Z 519.064,A -85,B 0,C 180,E1 -7463.084,E2 -7463.084} C_VEL
LIN {X 0,Y 467.098,Z 514.232,A -85,B 0,C 180,E1 -7464.388,E2 -7464.388} C_VEL
LIN {X 0,Y 467.456,Z 507.282,A -85,B 0,C 180,E1 -7465.905,E2 -7465.905} C_VEL
LIN {X 0,Y 467.92,Z 498.708,A -85,B 0,C 180,E1 -7467.418,E2 -7467.418} C_VEL
LIN {X 0,Y 468.43,Z 489.772,A -85,B 0,C 180,E1 -7468.711,E2 -7468.711} C_VEL
LIN {X 0,Y 469.08,Z 478.984,A -85,B 0,C 180,E1 -7470,E2 -7470} C_VEL
LIN {X 0,Y 469.768,Z 468.041,A -85,B 0,C 180,E1 -7471.072,E2 -7471.072} C_VEL
LIN {X 0,Y 470.423,Z 456.038,A -85,B 0,C 180,E1 -7472.033,E2 -7472.033} C_VEL
LIN {X 0,Y 471.079,Z 442.615,A -85,B 0,C 180,E1 -7472.886,E2 -7472.886} C_VEL
LIN {X 0,Y 471.558,Z 429.674,A -85,B 0,C 180,E1 -7473.525,E2 -7473.525} C_VEL
LIN {X 0,Y 471.986,Z 414.835,A -85,B 0,C 180,E1 -7474.056,E2 -7474.056} C_VEL
LIN {X 0,Y 472.28,Z 401,A -85,B 0,C 180,E1 -7474.374,E2 -7474.374} C_VEL
LIN {X 0,Y 473.321,Z 286.594,A -85,B 0,C 180,E1 -7476.142,E2 -7476.142} C_VEL
LIN {X 0,Y 469.661,Z 269.161,A -85,B 0,C 180,E1 -7476.582,E2 -7476.582} C_VEL
LIN {X 0,Y 469.785,Z 260.68,A -85,B 0,C 180,E1 -7478.17,E2 -7478.17} C_VEL
LIN {X 0,Y 467.624,Z 249.864,A -85,B 0,C 180,E1 -7480.39,E2 -7480.39} C_VEL
LIN {X 0,Y 467.608,Z 249.863,A -85,B 0,C 180,E1 -7483.029,E2 -7483.029} C_VEL
LIN {X 0,Y 467.635,Z 249.863,A -85,B 0,C 180,E1 -7485.886,E2 -7485.886} C_VEL
LIN {X 0,Y 467.61,Z 249.86,A -85,B 0,C 180,E1 -7489.308,E2 -7489.308} C_VEL
LIN {X 0,Y 467.522,Z 249.872,A -85,B 0,C 180,E1 -7492.074,E2 -7492.074} C_VEL
LIN {X 0,Y 467.599,Z 249.86,A -85,B 0,C 180,E1 -7494.887,E2 -7494.887} C_VEL
LIN {X 0,Y 467.614,Z 249.864,A -85,B 0,C 180,E1 -7497.769,E2 -7497.769} C_VEL
